   1:  PR[91,2] = PR[90,2] + -10.552;
   1:L PR[91] R[100]mm/sec CNT100;
   1:  PR[91,1] = PR[90,1] + -1.730;
   1:  PR[91,2] = PR[90,2] + -9.704;
   1:L PR[91] R[100]mm/sec CNT100;
   1:  PR[91,1] = PR[90,1] + -0.458;
   1:  PR[91,2] = PR[90,2] + -9.382;
   1:L PR[91] R[100]mm/sec CNT100;
   1:  PR[91,1] = PR[90,1] + 0.617;
   1:L PR[91] R[100]mm/sec CNT100;
   1:  PR[91,1] = PR[90,1] + 1.895;
   1:  PR[91,2] = PR[90,2] + -9.703;
   1:L PR[91] R[100]mm/sec CNT100;
   1:  PR[91,1] = PR[90,1] + 2.818;
   1:  PR[91,2] = PR[90,2] + -10.551;
   1:L PR[91] R[100]mm/sec CNT100;
   1:  PR[91,1] = PR[90,1] + 4.830;
   1:  PR[91,2] = PR[90,2] + -13.079;
   1:L PR[91] R[100]mm/sec CNT100;
   1:  PR[91,1] = PR[90,1] + 7.355;
   1:  PR[91,2] = PR[90,2] + -15.363;
   1:L PR[91] R[100]mm/sec CNT100;
   1:  PR[91,1] = PR[90,1] + 9.557;
   1:  PR[91,2] = PR[90,2] + -16.817;
   1:L PR[91] R[100]mm/sec CNT100;
   1:  PR[91,1] = PR[90,1] + 10.825;
   1:  PR[91,2] = PR[90,2] + -17.449;
   1:L PR[91] R[100]mm/sec CNT100;
   1:  PR[91,1] = PR[90,1] + 12.898;
   1:  PR[91,2] = PR[90,2] + -18.381;
   1:L PR[91] R[100]mm/sec CNT100;
   1:  PR[91,1] = PR[90,1] + 15.573;
   1:  PR[91,2] = PR[90,2] + -19.015;
   1:L PR[91] R[100]mm/sec CNT100;
   1:  PR[91,1] = PR[90,1] + 17.209;
   1:  PR[91,2] = PR[90,2] + -19.446;
   1:L PR[91] R[100]mm/sec CNT100;
   1:  PR[91,1] = PR[90,1] + 18.228;
   1:  PR[91,2] = PR[90,2] + -19.564;
   1:L PR[91] R[100]mm/sec CNT100;
   1:  PR[91,1] = PR[90,1] + 22.320;
   1:  PR[91,2] = PR[90,2] + -19.544;
   1:L PR[91] R[100]mm/sec CNT100;
   1:  PR[91,1] = PR[90,1] + 22.708;
   1:  PR[91,2] = PR[90,2] + -19.528;
   1:L PR[91] R[100]mm/sec CNT100;
   1:  PR[91,1] = PR[90,1] + 27.496;
   1:  PR[91,2] = PR[90,2] + -18.402;
   1:L PR[91] R[100]mm/sec CNT100;
   1:  PR[91,1] = PR[90,1] + 31.736;
   1:  PR[91,2] = PR[90,2] + -16.280;
   1:L PR[91] R[100]mm/sec CNT100;
   1:  PR[91,1] = PR[90,1] + 32.455;
   1:  PR[91,2] = PR[90,2] + -15.698;
   1:L PR[91] R[100]mm/sec CNT100;
   1:  PR[91,1] = PR[90,1] + 35.347;
   1:  PR[91,2] = PR[90,2] + -13.226;
   1:L PR[91] R[100]mm/sec CNT100;
   1:  PR[91,1] = PR[90,1] + 36.249;
   1:  PR[91,2] = PR[90,2] + -12.006;
   1:L PR[91] R[100]mm/sec CNT100;
   1:  PR[91,1] = PR[90,1] + 38.120;
   1:  PR[91,2] = PR[90,2] + -9.367;
   1:L PR[91] R[100]mm/sec CNT100;
   1:  PR[91,1] = PR[90,1] + 38.834;
   1:  PR[91,2] = PR[90,2] + -7.622;
   1:L PR[91] R[100]mm/sec CNT100;
   1:  PR[91,1] = PR[90,1] + 39.865;
   1:  PR[91,2] = PR[90,2] + -5.033;
   1:L PR[91] R[100]mm/sec CNT100;
   1:  PR[91,1] = PR[90,1] + 40.172;
   1:  PR[91,2] = PR[90,2] + -2.721;
   1:L PR[91] R[100]mm/sec CNT100;
   1:  PR[91,1] = PR[90,1] + 40.468;
   1:  PR[91,2] = PR[90,2] + -0.320;
   1:L PR[91] R[100]mm/sec CNT100;
   1:  PR[91,1] = PR[90,1] + 40.178;
   1:  PR[91,2] = PR[90,2] + 1.844;
   1:L PR[91] R[100]mm/sec CNT100;
   1:  PR[91,1] = PR[90,1] + 39.862;
   1:  PR[91,2] = PR[90,2] + 4.417;
   1:L PR[91] R[100]mm/sec CNT100;
   1:  PR[91,1] = PR[90,1] + 38.833;
   1:  PR[91,2] = PR[90,2] + 7.000;
   1:L PR[91] R[100]mm/sec CNT100;
   1:  PR[91,1] = PR[90,1] + 38.120;
   1:  PR[91,2] = PR[90,2] + 8.744;
   1:L PR[91] R[100]mm/sec CNT100;
   1:  PR[91,1] = PR[90,1] + 36.247;
   1:  PR[91,2] = PR[90,2] + 11.384;
   1:L PR[91] R[100]mm/sec CNT100;
   1:  PR[91,1] = PR[90,1] + 35.345;
   1:  PR[91,2] = PR[90,2] + 12.604;
   1:L PR[91] R[100]mm/sec CNT100;
   1:  PR[91,1] = PR[90,1] + 32.451;
   1:  PR[91,2] = PR[90,2] + 15.077;
   1:L PR[91] R[100]mm/sec CNT100;
   1:  PR[91,1] = PR[90,1] + 31.733;
   1:  PR[91,2] = PR[90,2] + 15.658;
   1:L PR[91] R[100]mm/sec CNT100;
   1:  PR[91,1] = PR[90,1] + 27.488;
   1:  PR[91,2] = PR[90,2] + 17.781;
   1:L PR[91] R[100]mm/sec CNT100;
   1:  PR[91,1] = PR[90,1] + 22.979;
   1:  PR[91,2] = PR[90,2] + 18.854;
   1:L PR[91] R[100]mm/sec CNT100;
   1:  PR[91,1] = PR[90,1] + 22.725;
   1:  PR[91,2] = PR[90,2] + 18.904;
   1:L PR[91] R[100]mm/sec CNT100;
   1:  PR[91,1] = PR[90,1] + 22.312;
   1:  PR[91,2] = PR[90,2] + 18.921;
   1:L PR[91] R[100]mm/sec CNT100;
   1:  PR[91,1] = PR[90,1] + 18.222;
   1:  PR[91,2] = PR[90,2] + 18.939;
   1:L PR[91] R[100]mm/sec CNT100;
   1:  PR[91,1] = PR[90,1] + 17.181;
   1:  PR[91,2] = PR[90,2] + 18.819;
   1:L PR[91] R[100]mm/sec CNT100;
   1:  PR[91,1] = PR[90,1] + 14.439;
   1:  PR[91,2] = PR[90,2] + 18.179;
   1:L PR[91] R[100]mm/sec CNT100;
   1:  PR[91,1] = PR[90,1] + 12.914;
   1:  PR[91,2] = PR[90,2] + 17.765;
   1:L PR[91] R[100]mm/sec CNT100;
   1:  PR[91,1] = PR[90,1] + 10.821;
   1:  PR[91,2] = PR[90,2] + 16.824;
   1:L PR[91] R[100]mm/sec CNT100;
   1:  PR[91,1] = PR[90,1] + 9.555;
   1:  PR[91,2] = PR[90,2] + 16.191;
   1:L PR[91] R[100]mm/sec CNT100;
   1:  PR[91,1] = PR[90,1] + 7.337;
   1:  PR[91,2] = PR[90,2] + 14.727;
   1:L PR[91] R[100]mm/sec CNT100;
   1:  PR[91,1] = PR[90,1] + 6.997;
   1:  PR[91,2] = PR[90,2] + 14.436;
   1:L PR[91] R[100]mm/sec CNT100;
   1:  PR[91,1] = PR[90,1] + 4.838;
   1:  PR[91,2] = PR[90,2] + 12.463;
   1:L PR[91] R[100]mm/sec CNT100;
   1:  PR[91,1] = PR[90,1] + 2.867;
   1:  PR[91,2] = PR[90,2] + 9.964;
   1:L PR[91] R[100]mm/sec CNT100;
   1:  PR[91,1] = PR[90,1] + 1.892;
   1:  PR[91,2] = PR[90,2] + 9.079;
   1:L PR[91] R[100]mm/sec CNT100;
   1:  PR[91,1] = PR[90,1] + 0.623;
   1:  PR[91,2] = PR[90,2] + 8.758;
   1:L PR[91] R[100]mm/sec CNT100;
   1:  PR[91,1] = PR[90,1] + -0.452;
   1:L PR[91] R[100]mm/sec CNT100;
   1:  PR[91] = PR[90];
   1:  PR[91,1] = PR[90,1] + -1.625;
   1:  PR[91,2] = PR[90,2] + 9.360;
   1:  PR[91,3] = PR[90,3] + 22.875;
   1:L PR[91] R[100]mm/sec CNT100;
   1:  PR[91,1] = PR[90,1] + -2.543;
   1:  PR[91,2] = PR[90,2] + 10.196;
   1:L PR[91] R[100]mm/sec CNT100;
   1:  PR[91,1] = PR[90,1] + -4.007;
   1:  PR[91,2] = PR[90,2] + 12.033;
   1:L PR[91] R[100]mm/sec CNT100;
   1:  PR[91,1] = PR[90,1] + -4.437;
   1:  PR[91,2] = PR[90,2] + 12.534;
   1:L PR[91] R[100]mm/sec CNT100;
   1:  PR[91,1] = PR[90,1] + -6.783;
   1:  PR[91,2] = PR[90,2] + 14.646;
   1:L PR[91] R[100]mm/sec CNT100;
   1:  PR[91,1] = PR[90,1] + -9.375;
   1:  PR[91,2] = PR[90,2] + 16.350;
   1:L PR[91] R[100]mm/sec CNT100;
   1:  PR[91,1] = PR[90,1] + -9.956;
   1:  PR[91,2] = PR[90,2] + 16.641;
   1:L PR[91] R[100]mm/sec CNT100;
   1:  PR[91,1] = PR[90,1] + -12.537;
   1:  PR[91,2] = PR[90,2] + 17.804;
   1:L PR[91] R[100]mm/sec CNT100;
   1:  PR[91,1] = PR[90,1] + -14.370;
   1:  PR[91,2] = PR[90,2] + 18.238;
   1:L PR[91] R[100]mm/sec CNT100;
   1:  PR[91,1] = PR[90,1] + -16.616;
   1:  PR[91,2] = PR[90,2] + 18.828;
   1:L PR[91] R[100]mm/sec CNT100;
   1:  PR[91,1] = PR[90,1] + -18.071;
   1:  PR[91,2] = PR[90,2] + 18.995;
   1:L PR[91] R[100]mm/sec CNT100;
   1:  PR[91,1] = PR[90,1] + -21.480;
   1:  PR[91,2] = PR[90,2] + 18.979;
   1:L PR[91] R[100]mm/sec CNT100;
   1:  PR[91,1] = PR[90,1] + -22.359;
   1:  PR[91,2] = PR[90,2] + 18.941;
   1:L PR[91] R[100]mm/sec CNT100;
   1:  PR[91,1] = PR[90,1] + -27.198;
   1:  PR[91,2] = PR[90,2] + 17.808;
   1:L PR[91] R[100]mm/sec CNT100;
   1:  PR[91,1] = PR[90,1] + -27.224;
   1:  PR[91,2] = PR[90,2] + 17.799;
   1:L PR[91] R[100]mm/sec CNT100;
   1:  PR[91,1] = PR[90,1] + -31.508;
   1:  PR[91,2] = PR[90,2] + 15.637;
   1:L PR[91] R[100]mm/sec CNT100;
   1:  PR[91,1] = PR[90,1] + -31.793;
   1:  PR[91,2] = PR[90,2] + 15.406;
   1:L PR[91] R[100]mm/sec CNT100;
   1:  PR[91,1] = PR[90,1] + -35.102;
   1:  PR[91,2] = PR[90,2] + 12.583;
   1:L PR[91] R[100]mm/sec CNT100;
   1:  PR[91,1] = PR[90,1] + -35.690;
   1:  PR[91,2] = PR[90,2] + 11.788;
   1:L PR[91] R[100]mm/sec CNT100;
   1:  PR[91,1] = PR[90,1] + -37.860;
   1:  PR[91,2] = PR[90,2] + 8.730;
   1:L PR[91] R[100]mm/sec CNT100;
   1:  PR[91,1] = PR[90,1] + -38.386;
   1:  PR[91,2] = PR[90,2] + 7.439;
   1:L PR[91] R[100]mm/sec CNT100;
   1:  PR[91,1] = PR[90,1] + -39.595;
   1:  PR[91,2] = PR[90,2] + 4.386;
   1:L PR[91] R[100]mm/sec CNT100;
   1:  PR[91,1] = PR[90,1] + -39.833;
   1:  PR[91,2] = PR[90,2] + 2.603;
   1:L PR[91] R[100]mm/sec CNT100;
   1:  PR[91,1] = PR[90,1] + -40.192;
   1:  PR[91,2] = PR[90,2] + -0.304;
   1:L PR[91] R[100]mm/sec CNT100;
   1:  PR[91,1] = PR[90,1] + -39.962;
   1:  PR[91,2] = PR[90,2] + -2.011;
   1:L PR[91] R[100]mm/sec CNT100;
   1:  PR[91,1] = PR[90,1] + -39.593;
   1:  PR[91,2] = PR[90,2] + -5.017;
   1:L PR[91] R[100]mm/sec CNT100;
   1:  PR[91,1] = PR[90,1] + -38.386;
   1:  PR[91,2] = PR[90,2] + -8.063;
   1:L PR[91] R[100]mm/sec CNT100;
   1:  PR[91,1] = PR[90,1] + -37.860;
   1:  PR[91,2] = PR[90,2] + -9.354;
   1:L PR[91] R[100]mm/sec CNT100;
   1:  PR[91,1] = PR[90,1] + -35.690;
   1:  PR[91,2] = PR[90,2] + -12.413;
   1:L PR[91] R[100]mm/sec CNT100;
   1:  PR[91,1] = PR[90,1] + -35.101;
   1:  PR[91,2] = PR[90,2] + -13.207;
   1:L PR[91] R[100]mm/sec CNT100;
   1:  PR[91,1] = PR[90,1] + -31.793;
   1:  PR[91,2] = PR[90,2] + -16.030;
   1:L PR[91] R[100]mm/sec CNT100;
   1:  PR[91,1] = PR[90,1] + -31.508;
   1:  PR[91,2] = PR[90,2] + -16.261;
   1:L PR[91] R[100]mm/sec CNT100;
   1:  PR[91,1] = PR[90,1] + -27.224;
   1:  PR[91,2] = PR[90,2] + -18.423;
   1:L PR[91] R[100]mm/sec CNT100;
   1:  PR[91,1] = PR[90,1] + -27.194;
   1:  PR[91,2] = PR[90,2] + -18.434;
   1:L PR[91] R[100]mm/sec CNT100;
   1:  PR[91,1] = PR[90,1] + -22.977;
   1:  PR[91,2] = PR[90,2] + -19.446;
   1:L PR[91] R[100]mm/sec CNT100;
   1:  PR[91,1] = PR[90,1] + -22.382;
   1:  PR[91,2] = PR[90,2] + -19.564;
   1:L PR[91] R[100]mm/sec CNT100;
   1:  PR[91,1] = PR[90,1] + -21.480;
   1:  PR[91,2] = PR[90,2] + -19.603;
   1:L PR[91] R[100]mm/sec CNT100;
   1:  PR[91,1] = PR[90,1] + -18.071;
   1:  PR[91,2] = PR[90,2] + -19.619;
   1:L PR[91] R[100]mm/sec CNT100;
   1:  PR[91,1] = PR[90,1] + -16.595;
   1:  PR[91,2] = PR[90,2] + -19.450;
   1:L PR[91] R[100]mm/sec CNT100;
   1:  PR[91,1] = PR[90,1] + -14.455;
   1:  PR[91,2] = PR[90,2] + -18.953;
   1:L PR[91] R[100]mm/sec CNT100;
   1:  PR[91,1] = PR[90,1] + -12.559;
   1:  PR[91,2] = PR[90,2] + -18.438;
   1:L PR[91] R[100]mm/sec CNT100;
   1:  PR[91,1] = PR[90,1] + -9.956;
   1:  PR[91,2] = PR[90,2] + -17.265;
   1:L PR[91] R[100]mm/sec CNT100;
   1:  PR[91,1] = PR[90,1] + -9.375;
   1:  PR[91,2] = PR[90,2] + -16.974;
   1:L PR[91] R[100]mm/sec CNT100;
   1:  PR[91,1] = PR[90,1] + -6.778;
   1:  PR[91,2] = PR[90,2] + -15.266;
   1:L PR[91] R[100]mm/sec CNT100;
   1:  PR[91,1] = PR[90,1] + -4.421;
   1:  PR[91,2] = PR[90,2] + -13.143;
   1:L PR[91] R[100]mm/sec CNT100;
   1:  PR[91,1] = PR[90,1] + -4.010;
   1:  PR[91,2] = PR[90,2] + -12.660;
   1:L PR[91] R[100]mm/sec CNT100;
   1:  PR[91,1] = PR[90,1] + -2.559;
   1:  PR[91,2] = PR[90,2] + -10.827;
   1:L PR[91] R[100]mm/sec CNT100;
   1:  PR[91,1] = PR[90,1] + -2.107;
   1:  PR[91,2] = PR[90,2] + -10.408;
   1:L PR[91] R[100]mm/sec CNT100;
   1:  PR[91,1] = PR[90,1] + -1.599;
   1:  PR[91,2] = PR[90,2] + -9.979;
   1:L PR[91] R[100]mm/sec CNT100;
   1:  PR[91,1] = PR[90,1] + -0.366;
   1:  PR[91,2] = PR[90,2] + -9.671;
   1:L PR[91] R[100]mm/sec CNT100;
   1:  PR[91,1] = PR[90,1] + 0.518;
   1:L PR[91] R[100]mm/sec CNT100;
   1:  PR[91,1] = PR[90,1] + 1.789;
   1:  PR[91,2] = PR[90,2] + -9.983;
   1:L PR[91] R[100]mm/sec CNT100;
   1:  PR[91,1] = PR[90,1] + 2.707;
   1:  PR[91,2] = PR[90,2] + -10.818;
   1:L PR[91] R[100]mm/sec CNT100;
   1:  PR[91,1] = PR[90,1] + 4.190;
   1:  PR[91,2] = PR[90,2] + -12.679;
   1:L PR[91] R[100]mm/sec CNT100;
   1:  PR[91,1] = PR[90,1] + 4.604;
   1:  PR[91,2] = PR[90,2] + -13.165;
   1:L PR[91] R[100]mm/sec CNT100;
   1:  PR[91,1] = PR[90,1] + 6.958;
   1:  PR[91,2] = PR[90,2] + -15.287;
   1:L PR[91] R[100]mm/sec CNT100;
   1:  PR[91,1] = PR[90,1] + 9.528;
   1:  PR[91,2] = PR[90,2] + -16.975;
   1:L PR[91] R[100]mm/sec CNT100;
   1:  PR[91,1] = PR[90,1] + 10.108;
   1:  PR[91,2] = PR[90,2] + -17.265;
   1:L PR[91] R[100]mm/sec CNT100;
   1:  PR[91,1] = PR[90,1] + 12.688;
   1:  PR[91,2] = PR[90,2] + -18.424;
   1:L PR[91] R[100]mm/sec CNT100;
   1:  PR[91,1] = PR[90,1] + 14.520;
   1:  PR[91,2] = PR[90,2] + -18.859;
   1:L PR[91] R[100]mm/sec CNT100;
   1:  PR[91,1] = PR[90,1] + 16.772;
   1:  PR[91,2] = PR[90,2] + -19.452;
   1:L PR[91] R[100]mm/sec CNT100;
   1:  PR[91,1] = PR[90,1] + 18.224;
   1:  PR[91,2] = PR[90,2] + -19.619;
   1:L PR[91] R[100]mm/sec CNT100;
   1:  PR[91,1] = PR[90,1] + 21.633;
   1:  PR[91,2] = PR[90,2] + -19.603;
   1:L PR[91] R[100]mm/sec CNT100;
   1:  PR[91,1] = PR[90,1] + 22.509;
   1:  PR[91,2] = PR[90,2] + -19.566;
   1:L PR[91] R[100]mm/sec CNT100;
   1:  PR[91,1] = PR[90,1] + 27.353;
   1:  PR[91,2] = PR[90,2] + -18.431;
   1:L PR[91] R[100]mm/sec CNT100;
   1:  PR[91,1] = PR[90,1] + 27.381;
   1:  PR[91,2] = PR[90,2] + -18.421;
   1:L PR[91] R[100]mm/sec CNT100;
   1:  PR[91,1] = PR[90,1] + 31.664;
   1:  PR[91,2] = PR[90,2] + -16.264;
   1:L PR[91] R[100]mm/sec CNT100;
   1:  PR[91,1] = PR[90,1] + 31.949;
   1:  PR[91,2] = PR[90,2] + -16.034;
   1:L PR[91] R[100]mm/sec CNT100;
   1:  PR[91,1] = PR[90,1] + 35.258;
   1:  PR[91,2] = PR[90,2] + -13.206;
   1:L PR[91] R[100]mm/sec CNT100;
   1:  PR[91,1] = PR[90,1] + 35.846;
   1:  PR[91,2] = PR[90,2] + -12.410;
   1:L PR[91] R[100]mm/sec CNT100;
   1:  PR[91,1] = PR[90,1] + 38.014;
   1:  PR[91,2] = PR[90,2] + -9.352;
   1:L PR[91] R[100]mm/sec CNT100;
   1:  PR[91,1] = PR[90,1] + 39.752;
   1:  PR[91,2] = PR[90,2] + -5.024;
   1:L PR[91] R[100]mm/sec CNT100;
   1:  PR[91,1] = PR[90,1] + 39.990;
   1:  PR[91,2] = PR[90,2] + -3.239;
   1:L PR[91] R[100]mm/sec CNT100;
   1:  PR[91,1] = PR[90,1] + 40.349;
   1:  PR[91,2] = PR[90,2] + -0.320;
   1:L PR[91] R[100]mm/sec CNT100;
   1:  PR[91,1] = PR[90,1] + 40.119;
   1:  PR[91,2] = PR[90,2] + 1.392;
   1:L PR[91] R[100]mm/sec CNT100;
   1:  PR[91,1] = PR[90,1] + 39.749;
   1:  PR[91,2] = PR[90,2] + 4.407;
   1:L PR[91] R[100]mm/sec CNT100;
   1:  PR[91,1] = PR[90,1] + 38.013;
   1:  PR[91,2] = PR[90,2] + 8.730;
   1:L PR[91] R[100]mm/sec CNT100;
   1:  PR[91,1] = PR[90,1] + 35.844;
   1:  PR[91,2] = PR[90,2] + 11.789;
   1:L PR[91] R[100]mm/sec CNT100;
   1:  PR[91,1] = PR[90,1] + 35.256;
   1:  PR[91,2] = PR[90,2] + 12.584;
   1:L PR[91] R[100]mm/sec CNT100;
   1:  PR[91,1] = PR[90,1] + 31.944;
   1:  PR[91,2] = PR[90,2] + 15.413;
   1:L PR[91] R[100]mm/sec CNT100;
   1:  PR[91,1] = PR[90,1] + 31.660;
   1:  PR[91,2] = PR[90,2] + 15.643;
   1:L PR[91] R[100]mm/sec CNT100;
   1:  PR[91,1] = PR[90,1] + 27.374;
   1:  PR[91,2] = PR[90,2] + 17.799;
   1:L PR[91] R[100]mm/sec CNT100;
   1:  PR[91,1] = PR[90,1] + 27.343;
   1:  PR[91,2] = PR[90,2] + 17.811;
   1:L PR[91] R[100]mm/sec CNT100;
   1:  PR[91,1] = PR[90,1] + 23.123;
   1:  PR[91,2] = PR[90,2] + 18.824;
   1:L PR[91] R[100]mm/sec CNT100;
   1:  PR[91,1] = PR[90,1] + 22.527;
   1:  PR[91,2] = PR[90,2] + 18.942;
   1:L PR[91] R[100]mm/sec CNT100;
   1:  PR[91,1] = PR[90,1] + 21.627;
   1:  PR[91,2] = PR[90,2] + 18.980;
   1:L PR[91] R[100]mm/sec CNT100;
   1:  PR[91,1] = PR[90,1] + 18.218;
   1:  PR[91,2] = PR[90,2] + 18.994;
   1:L PR[91] R[100]mm/sec CNT100;
   1:  PR[91,1] = PR[90,1] + 16.746;
   1:  PR[91,2] = PR[90,2] + 18.825;
   1:L PR[91] R[100]mm/sec CNT100;
   1:  PR[91,1] = PR[90,1] + 14.607;
   1:  PR[91,2] = PR[90,2] + 18.326;
   1:L PR[91] R[100]mm/sec CNT100;
   1:  PR[91,1] = PR[90,1] + 12.706;
   1:  PR[91,2] = PR[90,2] + 17.808;
   1:L PR[91] R[100]mm/sec CNT100;
   1:  PR[91,1] = PR[90,1] + 10.107;
   1:  PR[91,2] = PR[90,2] + 16.640;
   1:L PR[91] R[100]mm/sec CNT100;
   1:  PR[91,1] = PR[90,1] + 9.527;
   1:  PR[91,2] = PR[90,2] + 16.351;
   1:L PR[91] R[100]mm/sec CNT100;
   1:  PR[91,1] = PR[90,1] + 6.962;
   1:  PR[91,2] = PR[90,2] + 14.667;
   1:L PR[91] R[100]mm/sec CNT100;
   1:  PR[91,1] = PR[90,1] + 4.591;
   1:  PR[91,2] = PR[90,2] + 12.531;
   1:L PR[91] R[100]mm/sec CNT100;
   1:  PR[91,1] = PR[90,1] + 4.554;
   1:  PR[91,2] = PR[90,2] + 12.492;
   1:L PR[91] R[100]mm/sec CNT100;
   1:  PR[91,1] = PR[90,1] + 2.769;
   1:  PR[91,2] = PR[90,2] + 10.224;
   1:L PR[91] R[100]mm/sec CNT100;
   1:  PR[91,1] = PR[90,1] + 2.592;
   1:  PR[91,2] = PR[90,2] + 10.088;
   1:L PR[91] R[100]mm/sec CNT100;
   1:  PR[91,1] = PR[90,1] + 2.279;
   1:  PR[91,2] = PR[90,2] + 9.789;
   1:L PR[91] R[100]mm/sec CNT100;
   1:  PR[91,1] = PR[90,1] + 1.763;
   1:  PR[91,2] = PR[90,2] + 9.354;
   1:L PR[91] R[100]mm/sec CNT100;
   1:  PR[91,1] = PR[90,1] + 0.530;
   1:  PR[91,2] = PR[90,2] + 9.047;
   1:L PR[91] R[100]mm/sec CNT100;
   1:  PR[91,1] = PR[90,1] + -0.352;
   1:L PR[91] R[100]mm/sec CNT100;
   1:  PR[91] = PR[90];
   1:  PR[91,1] = PR[90,1] + -1.514;
   1:  PR[91,2] = PR[90,2] + 9.639;
   1:  PR[91,3] = PR[90,3] + 23.485;
   1:L PR[91] R[100]mm/sec CNT100;
   1:  PR[91,1] = PR[90,1] + -2.434;
   1:  PR[91,2] = PR[90,2] + 10.459;
   1:L PR[91] R[100]mm/sec CNT100;
   1:  PR[91,1] = PR[90,1] + -3.410;
   1:  PR[91,2] = PR[90,2] + 11.680;
   1:L PR[91] R[100]mm/sec CNT100;
   1:  PR[91,1] = PR[90,1] + -4.067;
   1:  PR[91,2] = PR[90,2] + 12.470;
   1:L PR[91] R[100]mm/sec CNT100;
   1:  PR[91,1] = PR[90,1] + -4.215;
   1:  PR[91,2] = PR[90,2] + 12.625;
   1:L PR[91] R[100]mm/sec CNT100;
   1:  PR[91,1] = PR[90,1] + -6.555;
   1:  PR[91,2] = PR[90,2] + 14.723;
   1:L PR[91] R[100]mm/sec CNT100;
   1:  PR[91,1] = PR[90,1] + -9.313;
   1:  PR[91,2] = PR[90,2] + 16.490;
   1:L PR[91] R[100]mm/sec CNT100;
   1:  PR[91,1] = PR[90,1] + -12.328;
   1:  PR[91,2] = PR[90,2] + 17.848;
   1:L PR[91] R[100]mm/sec CNT100;
   1:  PR[91,1] = PR[90,1] + -13.319;
   1:  PR[91,2] = PR[90,2] + 18.083;
   1:L PR[91] R[100]mm/sec CNT100;
   1:  PR[91,1] = PR[90,1] + -16.179;
   1:  PR[91,2] = PR[90,2] + 18.834;
   1:L PR[91] R[100]mm/sec CNT100;
   1:  PR[91,1] = PR[90,1] + -18.067;
   1:  PR[91,2] = PR[90,2] + 19.050;
   1:L PR[91] R[100]mm/sec CNT100;
   1:  PR[91,1] = PR[90,1] + -20.795;
   1:  PR[91,2] = PR[90,2] + 19.037;
   1:L PR[91] R[100]mm/sec CNT100;
   1:  PR[91,1] = PR[90,1] + -22.161;
   1:  PR[91,2] = PR[90,2] + 18.979;
   1:L PR[91] R[100]mm/sec CNT100;
   1:  PR[91,1] = PR[90,1] + -26.109;
   1:  PR[91,2] = PR[90,2] + 18.049;
   1:L PR[91] R[100]mm/sec CNT100;
   1:  PR[91,1] = PR[90,1] + -26.826;
   1:  PR[91,2] = PR[90,2] + 17.900;
   1:L PR[91] R[100]mm/sec CNT100;
   1:  PR[91,1] = PR[90,1] + -27.197;
   1:  PR[91,2] = PR[90,2] + 17.765;
   1:L PR[91] R[100]mm/sec CNT100;
   1:  PR[91,1] = PR[90,1] + -31.416;
   1:  PR[91,2] = PR[90,2] + 15.631;
   1:L PR[91] R[100]mm/sec CNT100;
   1:  PR[91,1] = PR[90,1] + -35.012;
   1:  PR[91,2] = PR[90,2] + 12.563;
   1:L PR[91] R[100]mm/sec CNT100;
   1:  PR[91,1] = PR[90,1] + -35.287;
   1:  PR[91,2] = PR[90,2] + 12.192;
   1:L PR[91] R[100]mm/sec CNT100;
   1:  PR[91,1] = PR[90,1] + -37.753;
   1:  PR[91,2] = PR[90,2] + 8.716;
   1:L PR[91] R[100]mm/sec CNT100;
   1:  PR[91,1] = PR[90,1] + -39.482;
   1:  PR[91,2] = PR[90,2] + 4.377;
   1:L PR[91] R[100]mm/sec CNT100;
   1:  PR[91,1] = PR[90,1] + -39.650;
   1:  PR[91,2] = PR[90,2] + 3.118;
   1:L PR[91] R[100]mm/sec CNT100;
   1:  PR[91,1] = PR[90,1] + -40.073;
   1:  PR[91,2] = PR[90,2] + -0.304;
   1:L PR[91] R[100]mm/sec CNT100;
   1:  PR[91,1] = PR[90,1] + -39.904;
   1:  PR[91,2] = PR[90,2] + -1.560;
   1:L PR[91] R[100]mm/sec CNT100;
   1:  PR[91,1] = PR[90,1] + -39.479;
   1:  PR[91,2] = PR[90,2] + -5.009;
   1:L PR[91] R[100]mm/sec CNT100;
   1:  PR[91,1] = PR[90,1] + -38.095;
   1:  PR[91,2] = PR[90,2] + -8.505;
   1:L PR[91] R[100]mm/sec CNT100;
   1:  PR[91,1] = PR[90,1] + -37.756;
   1:  PR[91,2] = PR[90,2] + -9.336;
   1:L PR[91] R[100]mm/sec CNT100;
   1:  PR[91,1] = PR[90,1] + -35.286;
   1:  PR[91,2] = PR[90,2] + -12.816;
   1:L PR[91] R[100]mm/sec CNT100;
   1:  PR[91,1] = PR[90,1] + -35.012;
   1:  PR[91,2] = PR[90,2] + -13.187;
   1:L PR[91] R[100]mm/sec CNT100;
   1:  PR[91,1] = PR[90,1] + -31.415;
   1:  PR[91,2] = PR[90,2] + -16.255;
   1:L PR[91] R[100]mm/sec CNT100;
   1:  PR[91,1] = PR[90,1] + -27.197;
   1:  PR[91,2] = PR[90,2] + -18.389;
   1:L PR[91] R[100]mm/sec CNT100;
   1:  PR[91,1] = PR[90,1] + -26.805;
   1:  PR[91,2] = PR[90,2] + -18.532;
   1:L PR[91] R[100]mm/sec CNT100;
   1:  PR[91,1] = PR[90,1] + -23.123;
   1:  PR[91,2] = PR[90,2] + -19.415;
   1:L PR[91] R[100]mm/sec CNT100;
   1:  PR[91,1] = PR[90,1] + -22.186;
   1:  PR[91,2] = PR[90,2] + -19.602;
   1:L PR[91] R[100]mm/sec CNT100;
   1:  PR[91,1] = PR[90,1] + -20.795;
   1:  PR[91,2] = PR[90,2] + -19.661;
   1:L PR[91] R[100]mm/sec CNT100;
   1:  PR[91,1] = PR[90,1] + -18.067;
   1:  PR[91,2] = PR[90,2] + -19.674;
   1:L PR[91] R[100]mm/sec CNT100;
   1:  PR[91,1] = PR[90,1] + -16.159;
   1:  PR[91,2] = PR[90,2] + -19.455;
   1:L PR[91] R[100]mm/sec CNT100;
   1:  PR[91,1] = PR[90,1] + -14.622;
   1:  PR[91,2] = PR[90,2] + -19.099;
   1:L PR[91] R[100]mm/sec CNT100;
   1:  PR[91,1] = PR[90,1] + -12.350;
   1:  PR[91,2] = PR[90,2] + -18.482;
   1:L PR[91] R[100]mm/sec CNT100;
   1:  PR[91,1] = PR[90,1] + -9.313;
   1:  PR[91,2] = PR[90,2] + -17.113;
   1:L PR[91] R[100]mm/sec CNT100;
   1:  PR[91,1] = PR[90,1] + -6.576;
   1:  PR[91,2] = PR[90,2] + -15.363;
   1:L PR[91] R[100]mm/sec CNT100;
   1:  PR[91,1] = PR[90,1] + -6.379;
   1:  PR[91,2] = PR[90,2] + -15.198;
   1:L PR[91] R[100]mm/sec CNT100;
   1:  PR[91,1] = PR[90,1] + -4.216;
   1:  PR[91,2] = PR[90,2] + -13.248;
   1:L PR[91] R[100]mm/sec CNT100;
   1:  PR[91,1] = PR[90,1] + -3.407;
   1:  PR[91,2] = PR[90,2] + -12.300;
   1:L PR[91] R[100]mm/sec CNT100;
   1:  PR[91,1] = PR[90,1] + -2.456;
   1:  PR[91,2] = PR[90,2] + -11.098;
   1:L PR[91] R[100]mm/sec CNT100;
   1:  PR[91,1] = PR[90,1] + -2.127;
   1:  PR[91,2] = PR[90,2] + -10.792;
   1:L PR[91] R[100]mm/sec CNT100;
   1:  PR[91,1] = PR[90,1] + -1.497;
   1:  PR[91,2] = PR[90,2] + -10.260;
   1:L PR[91] R[100]mm/sec CNT100;
   1:  PR[91,1] = PR[90,1] + -0.273;
   1:  PR[91,2] = PR[90,2] + -9.959;
   1:L PR[91] R[100]mm/sec CNT100;
   1:  PR[91,1] = PR[90,1] + 0.424;
   1:L PR[91] R[100]mm/sec CNT100;
   1:  PR[91,1] = PR[90,1] + 1.678;
   1:  PR[91,2] = PR[90,2] + -10.263;
   1:L PR[91] R[100]mm/sec CNT100;
   1:  PR[91,1] = PR[90,1] + 2.600;
   1:  PR[91,2] = PR[90,2] + -11.082;
   1:L PR[91] R[100]mm/sec CNT100;
   1:  PR[91,1] = PR[90,1] + 3.581;
   1:  PR[91,2] = PR[90,2] + -12.311;
   1:L PR[91] R[100]mm/sec CNT100;
   1:  PR[91,1] = PR[90,1] + 4.395;
   1:  PR[91,2] = PR[90,2] + -13.268;
   1:L PR[91] R[100]mm/sec CNT100;
   1:  PR[91,1] = PR[90,1] + 6.705;
   1:  PR[91,2] = PR[90,2] + -15.346;
   1:L PR[91] R[100]mm/sec CNT100;
   1:  PR[91,1] = PR[90,1] + 9.466;
   1:  PR[91,2] = PR[90,2] + -17.114;
   1:L PR[91] R[100]mm/sec CNT100;
   1:  PR[91,1] = PR[90,1] + 12.477;
   1:  PR[91,2] = PR[90,2] + -18.467;
   1:L PR[91] R[100]mm/sec CNT100;
   1:  PR[91,1] = PR[90,1] + 13.467;
   1:  PR[91,2] = PR[90,2] + -18.702;
   1:L PR[91] R[100]mm/sec CNT100;
   1:  PR[91,1] = PR[90,1] + 16.335;
   1:  PR[91,2] = PR[90,2] + -19.457;
   1:L PR[91] R[100]mm/sec CNT100;
   1:  PR[91,1] = PR[90,1] + 18.219;
   1:  PR[91,2] = PR[90,2] + -19.674;
   1:L PR[91] R[100]mm/sec CNT100;
   1:  PR[91,1] = PR[90,1] + 20.947;
   1:  PR[91,2] = PR[90,2] + -19.661;
   1:L PR[91] R[100]mm/sec CNT100;
   1:  PR[91,1] = PR[90,1] + 22.309;
   1:  PR[91,2] = PR[90,2] + -19.604;
   1:L PR[91] R[100]mm/sec CNT100;
   1:  PR[91,1] = PR[90,1] + 26.258;
   1:  PR[91,2] = PR[90,2] + -18.673;
   1:L PR[91] R[100]mm/sec CNT100;
   1:  PR[91,1] = PR[90,1] + 26.979;
   1:  PR[91,2] = PR[90,2] + -18.523;
   1:L PR[91] R[100]mm/sec CNT100;
   1:  PR[91,1] = PR[90,1] + 27.352;
   1:  PR[91,2] = PR[90,2] + -18.388;
   1:L PR[91] R[100]mm/sec CNT100;
   1:  PR[91,1] = PR[90,1] + 31.572;
   1:  PR[91,2] = PR[90,2] + -16.258;
   1:L PR[91] R[100]mm/sec CNT100;
   1:  PR[91,1] = PR[90,1] + 35.168;
   1:  PR[91,2] = PR[90,2] + -13.185;
   1:L PR[91] R[100]mm/sec CNT100;
   1:  PR[91,1] = PR[90,1] + 35.443;
   1:  PR[91,2] = PR[90,2] + -12.814;
   1:L PR[91] R[100]mm/sec CNT100;
   1:  PR[91,1] = PR[90,1] + 37.910;
   1:  PR[91,2] = PR[90,2] + -9.335;
   1:L PR[91] R[100]mm/sec CNT100;
   1:  PR[91,1] = PR[90,1] + 39.639;
   1:  PR[91,2] = PR[90,2] + -5.017;
   1:L PR[91] R[100]mm/sec CNT100;
   1:  PR[91,1] = PR[90,1] + 39.807;
   1:  PR[91,2] = PR[90,2] + -3.756;
   1:L PR[91] R[100]mm/sec CNT100;
   1:  PR[91,1] = PR[90,1] + 40.229;
   1:  PR[91,2] = PR[90,2] + -0.320;
   1:L PR[91] R[100]mm/sec CNT100;
   1:  PR[91,1] = PR[90,1] + 40.061;
   1:  PR[91,2] = PR[90,2] + 0.940;
   1:L PR[91] R[100]mm/sec CNT100;
   1:  PR[91,1] = PR[90,1] + 39.636;
   1:  PR[91,2] = PR[90,2] + 4.401;
   1:L PR[91] R[100]mm/sec CNT100;
   1:  PR[91,1] = PR[90,1] + 37.909;
   1:  PR[91,2] = PR[90,2] + 8.712;
   1:L PR[91] R[100]mm/sec CNT100;
   1:  PR[91,1] = PR[90,1] + 35.440;
   1:  PR[91,2] = PR[90,2] + 12.193;
   1:L PR[91] R[100]mm/sec CNT100;
   1:  PR[91,1] = PR[90,1] + 35.166;
   1:  PR[91,2] = PR[90,2] + 12.564;
   1:L PR[91] R[100]mm/sec CNT100;
   1:  PR[91,1] = PR[90,1] + 31.567;
   1:  PR[91,2] = PR[90,2] + 15.637;
   1:L PR[91] R[100]mm/sec CNT100;
   1:  PR[91,1] = PR[90,1] + 27.346;
   1:  PR[91,2] = PR[90,2] + 17.766;
   1:L PR[91] R[100]mm/sec CNT100;
   1:  PR[91,1] = PR[90,1] + 26.951;
   1:  PR[91,2] = PR[90,2] + 17.909;
   1:L PR[91] R[100]mm/sec CNT100;
   1:  PR[91,1] = PR[90,1] + 23.267;
   1:  PR[91,2] = PR[90,2] + 18.794;
   1:L PR[91] R[100]mm/sec CNT100;
   1:  PR[91,1] = PR[90,1] + 22.329;
   1:  PR[91,2] = PR[90,2] + 18.980;
   1:L PR[91] R[100]mm/sec CNT100;
   1:  PR[91,1] = PR[90,1] + 20.941;
   1:  PR[91,2] = PR[90,2] + 19.038;
   1:L PR[91] R[100]mm/sec CNT100;
   1:  PR[91,1] = PR[90,1] + 18.214;
   1:  PR[91,2] = PR[90,2] + 19.050;
   1:L PR[91] R[100]mm/sec CNT100;
   1:  PR[91,1] = PR[90,1] + 16.310;
   1:  PR[91,2] = PR[90,2] + 18.830;
   1:L PR[91] R[100]mm/sec CNT100;
   1:  PR[91,1] = PR[90,1] + 14.775;
   1:  PR[91,2] = PR[90,2] + 18.472;
   1:L PR[91] R[100]mm/sec CNT100;
   1:  PR[91,1] = PR[90,1] + 12.497;
   1:  PR[91,2] = PR[90,2] + 17.852;
   1:L PR[91] R[100]mm/sec CNT100;
   1:  PR[91,1] = PR[90,1] + 9.466;
   1:  PR[91,2] = PR[90,2] + 16.490;
   1:L PR[91] R[100]mm/sec CNT100;
   1:  PR[91,1] = PR[90,1] + 6.734;
   1:  PR[91,2] = PR[90,2] + 14.743;
   1:L PR[91] R[100]mm/sec CNT100;
   1:  PR[91,1] = PR[90,1] + 4.396;
   1:  PR[91,2] = PR[90,2] + 12.646;
   1:L PR[91] R[100]mm/sec CNT100;
   1:  PR[91,1] = PR[90,1] + 4.260;
   1:  PR[91,2] = PR[90,2] + 12.504;
   1:L PR[91] R[100]mm/sec CNT100;
   1:  PR[91,1] = PR[90,1] + 2.742;
   1:  PR[91,2] = PR[90,2] + 10.574;
   1:L PR[91] R[100]mm/sec CNT100;
   1:  PR[91,1] = PR[90,1] + 2.284;
   1:  PR[91,2] = PR[90,2] + 10.161;
   1:L PR[91] R[100]mm/sec CNT100;
   1:  PR[91,1] = PR[90,1] + 1.661;
   1:  PR[91,2] = PR[90,2] + 9.636;
   1:L PR[91] R[100]mm/sec CNT100;
   1:  PR[91,1] = PR[90,1] + 0.437;
   1:  PR[91,2] = PR[90,2] + 9.335;
   1:L PR[91] R[100]mm/sec CNT100;
   1:  PR[91,1] = PR[90,1] + -0.258;
   1:L PR[91] R[100]mm/sec CNT100;
   1:  PR[91] = PR[90];
   1:  PR[91,1] = PR[90,1] + -1.401;
   1:  PR[91,2] = PR[90,2] + 9.919;
   1:  PR[91,3] = PR[90,3] + 24.095;
   1:L PR[91] R[100]mm/sec CNT100;
   1:  PR[91,1] = PR[90,1] + -2.322;
   1:  PR[91,2] = PR[90,2] + 10.715;
   1:L PR[91] R[100]mm/sec CNT100;
   1:  PR[91,1] = PR[90,1] + -3.778;
   1:  PR[91,2] = PR[90,2] + 12.487;
   1:L PR[91] R[100]mm/sec CNT100;
   1:  PR[91,1] = PR[90,1] + -4.025;
   1:  PR[91,2] = PR[90,2] + 12.745;
   1:L PR[91] R[100]mm/sec CNT100;
   1:  PR[91,1] = PR[90,1] + -6.030;
   1:  PR[91,2] = PR[90,2] + 14.552;
   1:L PR[91] R[100]mm/sec CNT100;
   1:  PR[91,1] = PR[90,1] + -6.319;
   1:  PR[91,2] = PR[90,2] + 14.797;
   1:L PR[91] R[100]mm/sec CNT100;
   1:  PR[91,1] = PR[90,1] + -9.021;
   1:  PR[91,2] = PR[90,2] + 16.529;
   1:L PR[91] R[100]mm/sec CNT100;
   1:  PR[91,1] = PR[90,1] + -12.128;
   1:  PR[91,2] = PR[90,2] + 17.897;
   1:L PR[91] R[100]mm/sec CNT100;
   1:  PR[91,1] = PR[90,1] + -15.741;
   1:  PR[91,2] = PR[90,2] + 18.839;
   1:L PR[91] R[100]mm/sec CNT100;
   1:  PR[91,1] = PR[90,1] + -18.064;
   1:  PR[91,2] = PR[90,2] + 19.105;
   1:L PR[91] R[100]mm/sec CNT100;
   1:  PR[91,1] = PR[90,1] + -20.110;
   1:  PR[91,2] = PR[90,2] + 19.096;
   1:L PR[91] R[100]mm/sec CNT100;
   1:  PR[91,1] = PR[90,1] + -21.964;
   1:  PR[91,2] = PR[90,2] + 19.017;
   1:L PR[91] R[100]mm/sec CNT100;
   1:  PR[91,1] = PR[90,1] + -25.192;
   1:  PR[91,2] = PR[90,2] + 18.256;
   1:L PR[91] R[100]mm/sec CNT100;
   1:  PR[91,1] = PR[90,1] + -26.437;
   1:  PR[91,2] = PR[90,2] + 17.998;
   1:L PR[91] R[100]mm/sec CNT100;
   1:  PR[91,1] = PR[90,1] + -27.172;
   1:  PR[91,2] = PR[90,2] + 17.731;
   1:L PR[91] R[100]mm/sec CNT100;
   1:  PR[91,1] = PR[90,1] + -30.981;
   1:  PR[91,2] = PR[90,2] + 15.804;
   1:L PR[91] R[100]mm/sec CNT100;
   1:  PR[91,1] = PR[90,1] + -31.213;
   1:  PR[91,2] = PR[90,2] + 15.675;
   1:L PR[91] R[100]mm/sec CNT100;
   1:  PR[91,1] = PR[90,1] + -34.914;
   1:  PR[91,2] = PR[90,2] + 12.549;
   1:L PR[91] R[100]mm/sec CNT100;
   1:  PR[91,1] = PR[90,1] + -37.648;
   1:  PR[91,2] = PR[90,2] + 8.699;
   1:L PR[91] R[100]mm/sec CNT100;
   1:  PR[91,1] = PR[90,1] + -39.367;
   1:  PR[91,2] = PR[90,2] + 4.375;
   1:L PR[91] R[100]mm/sec CNT100;
   1:  PR[91,1] = PR[90,1] + -39.954;
   1:  PR[91,2] = PR[90,2] + -0.312;
   1:L PR[91] R[100]mm/sec CNT100;
   1:  PR[91,1] = PR[90,1] + -39.367;
   1:  PR[91,2] = PR[90,2] + -5.000;
   1:L PR[91] R[100]mm/sec CNT100;
   1:  PR[91,1] = PR[90,1] + -37.804;
   1:  PR[91,2] = PR[90,2] + -8.945;
   1:L PR[91] R[100]mm/sec CNT100;
   1:  PR[91,1] = PR[90,1] + -37.652;
   1:  PR[91,2] = PR[90,2] + -9.318;
   1:L PR[91] R[100]mm/sec CNT100;
   1:  PR[91,1] = PR[90,1] + -34.913;
   1:  PR[91,2] = PR[90,2] + -13.175;
   1:L PR[91] R[100]mm/sec CNT100;
   1:  PR[91,1] = PR[90,1] + -31.388;
   1:  PR[91,2] = PR[90,2] + -16.169;
   1:L PR[91] R[100]mm/sec CNT100;
   1:  PR[91,1] = PR[90,1] + -31.237;
   1:  PR[91,2] = PR[90,2] + -16.286;
   1:L PR[91] R[100]mm/sec CNT100;
   1:  PR[91,1] = PR[90,1] + -30.981;
   1:  PR[91,2] = PR[90,2] + -16.428;
   1:L PR[91] R[100]mm/sec CNT100;
   1:  PR[91,1] = PR[90,1] + -27.171;
   1:  PR[91,2] = PR[90,2] + -18.355;
   1:L PR[91] R[100]mm/sec CNT100;
   1:  PR[91,1] = PR[90,1] + -26.416;
   1:  PR[91,2] = PR[90,2] + -18.630;
   1:L PR[91] R[100]mm/sec CNT100;
   1:  PR[91,1] = PR[90,1] + -23.270;
   1:  PR[91,2] = PR[90,2] + -19.385;
   1:L PR[91] R[100]mm/sec CNT100;
   1:  PR[91,1] = PR[90,1] + -21.989;
   1:  PR[91,2] = PR[90,2] + -19.640;
   1:L PR[91] R[100]mm/sec CNT100;
   1:  PR[91,1] = PR[90,1] + -20.110;
   1:  PR[91,2] = PR[90,2] + -19.720;
   1:L PR[91] R[100]mm/sec CNT100;
   1:  PR[91,1] = PR[90,1] + -18.063;
   1:  PR[91,2] = PR[90,2] + -19.729;
   1:L PR[91] R[100]mm/sec CNT100;
   1:  PR[91,1] = PR[90,1] + -15.722;
   1:  PR[91,2] = PR[90,2] + -19.461;
   1:L PR[91] R[100]mm/sec CNT100;
   1:  PR[91,1] = PR[90,1] + -14.790;
   1:  PR[91,2] = PR[90,2] + -19.245;
   1:L PR[91] R[100]mm/sec CNT100;
   1:  PR[91,1] = PR[90,1] + -12.135;
   1:  PR[91,2] = PR[90,2] + -18.524;
   1:L PR[91] R[100]mm/sec CNT100;
   1:  PR[91,1] = PR[90,1] + -9.014;
   1:  PR[91,2] = PR[90,2] + -17.149;
   1:L PR[91] R[100]mm/sec CNT100;
   1:  PR[91,1] = PR[90,1] + -6.347;
   1:  PR[91,2] = PR[90,2] + -15.443;
   1:L PR[91] R[100]mm/sec CNT100;
   1:  PR[91,1] = PR[90,1] + -6.304;
   1:  PR[91,2] = PR[90,2] + -15.412;
   1:L PR[91] R[100]mm/sec CNT100;
   1:  PR[91,1] = PR[90,1] + -5.967;
   1:  PR[91,2] = PR[90,2] + -15.116;
   1:L PR[91] R[100]mm/sec CNT100;
   1:  PR[91,1] = PR[90,1] + -4.010;
   1:  PR[91,2] = PR[90,2] + -13.352;
   1:L PR[91] R[100]mm/sec CNT100;
   1:  PR[91,1] = PR[90,1] + -2.804;
   1:  PR[91,2] = PR[90,2] + -11.939;
   1:L PR[91] R[100]mm/sec CNT100;
   1:  PR[91,1] = PR[90,1] + -2.352;
   1:  PR[91,2] = PR[90,2] + -11.368;
   1:L PR[91] R[100]mm/sec CNT100;
   1:  PR[91,1] = PR[90,1] + -2.147;
   1:  PR[91,2] = PR[90,2] + -11.177;
   1:L PR[91] R[100]mm/sec CNT100;
   1:  PR[91,1] = PR[90,1] + -1.394;
   1:  PR[91,2] = PR[90,2] + -10.542;
   1:L PR[91] R[100]mm/sec CNT100;
   1:  PR[91,1] = PR[90,1] + -0.180;
   1:  PR[91,2] = PR[90,2] + -10.248;
   1:L PR[91] R[100]mm/sec CNT100;
   1:  PR[91,1] = PR[90,1] + 0.337;
   1:L PR[91] R[100]mm/sec CNT100;
   1:  PR[91,1] = PR[90,1] + 1.567;
   1:  PR[91,2] = PR[90,2] + -10.543;
   1:L PR[91] R[100]mm/sec CNT100;
   1:  PR[91,1] = PR[90,1] + 2.495;
   1:  PR[91,2] = PR[90,2] + -11.345;
   1:L PR[91] R[100]mm/sec CNT100;
   1:  PR[91,1] = PR[90,1] + 2.973;
   1:  PR[91,2] = PR[90,2] + -11.944;
   1:L PR[91] R[100]mm/sec CNT100;
   1:  PR[91,1] = PR[90,1] + 4.187;
   1:  PR[91,2] = PR[90,2] + -13.370;
   1:L PR[91] R[100]mm/sec CNT100;
   1:  PR[91,1] = PR[90,1] + 6.460;
   1:  PR[91,2] = PR[90,2] + -15.411;
   1:L PR[91] R[100]mm/sec CNT100;
   1:  PR[91,1] = PR[90,1] + 9.169;
   1:  PR[91,2] = PR[90,2] + -17.150;
   1:L PR[91] R[100]mm/sec CNT100;
   1:  PR[91,1] = PR[90,1] + 12.276;
   1:  PR[91,2] = PR[90,2] + -18.516;
   1:L PR[91] R[100]mm/sec CNT100;
   1:  PR[91,1] = PR[90,1] + 15.896;
   1:  PR[91,2] = PR[90,2] + -19.462;
   1:L PR[91] R[100]mm/sec CNT100;
   1:  PR[91,1] = PR[90,1] + 18.214;
   1:  PR[91,2] = PR[90,2] + -19.730;
   1:L PR[91] R[100]mm/sec CNT100;
   1:  PR[91,1] = PR[90,1] + 20.260;
   1:  PR[91,2] = PR[90,2] + -19.720;
   1:L PR[91] R[100]mm/sec CNT100;
   1:  PR[91,1] = PR[90,1] + 22.109;
   1:  PR[91,2] = PR[90,2] + -19.643;
   1:L PR[91] R[100]mm/sec CNT100;
   1:  PR[91,1] = PR[90,1] + 25.336;
   1:  PR[91,2] = PR[90,2] + -18.881;
   1:L PR[91] R[100]mm/sec CNT100;
   1:  PR[91,1] = PR[90,1] + 26.586;
   1:  PR[91,2] = PR[90,2] + -18.622;
   1:L PR[91] R[100]mm/sec CNT100;
   1:  PR[91,1] = PR[90,1] + 27.324;
   1:  PR[91,2] = PR[90,2] + -18.355;
   1:L PR[91] R[100]mm/sec CNT100;
   1:  PR[91,1] = PR[90,1] + 31.136;
   1:  PR[91,2] = PR[90,2] + -16.431;
   1:L PR[91] R[100]mm/sec CNT100;
   1:  PR[91,1] = PR[90,1] + 31.368;
   1:  PR[91,2] = PR[90,2] + -16.304;
   1:L PR[91] R[100]mm/sec CNT100;
   1:  PR[91,1] = PR[90,1] + 34.548;
   1:  PR[91,2] = PR[90,2] + -13.619;
   1:L PR[91] R[100]mm/sec CNT100;
   1:  PR[91,1] = PR[90,1] + 35.075;
   1:  PR[91,2] = PR[90,2] + -13.168;
   1:L PR[91] R[100]mm/sec CNT100;
   1:  PR[91,1] = PR[90,1] + 37.805;
   1:  PR[91,2] = PR[90,2] + -9.317;
   1:L PR[91] R[100]mm/sec CNT100;
   1:  PR[91,1] = PR[90,1] + 39.524;
   1:  PR[91,2] = PR[90,2] + -5.015;
   1:L PR[91] R[100]mm/sec CNT100;
   1:  PR[91,1] = PR[90,1] + 40.111;
   1:  PR[91,2] = PR[90,2] + -0.312;
   1:L PR[91] R[100]mm/sec CNT100;
   1:  PR[91,1] = PR[90,1] + 39.523;
   1:  PR[91,2] = PR[90,2] + 4.392;
   1:L PR[91] R[100]mm/sec CNT100;
   1:  PR[91,1] = PR[90,1] + 37.804;
   1:  PR[91,2] = PR[90,2] + 8.695;
   1:L PR[91] R[100]mm/sec CNT100;
   1:  PR[91,1] = PR[90,1] + 35.066;
   1:  PR[91,2] = PR[90,2] + 12.552;
   1:L PR[91] R[100]mm/sec CNT100;
   1:  PR[91,1] = PR[90,1] + 31.537;
   1:  PR[91,2] = PR[90,2] + 15.554;
   1:L PR[91] R[100]mm/sec CNT100;
   1:  PR[91,1] = PR[90,1] + 31.389;
   1:  PR[91,2] = PR[90,2] + 15.669;
   1:L PR[91] R[100]mm/sec CNT100;
   1:  PR[91,1] = PR[90,1] + 31.132;
   1:  PR[91,2] = PR[90,2] + 15.811;
   1:L PR[91] R[100]mm/sec CNT100;
   1:  PR[91,1] = PR[90,1] + 27.320;
   1:  PR[91,2] = PR[90,2] + 17.733;
   1:L PR[91] R[100]mm/sec CNT100;
   1:  PR[91,1] = PR[90,1] + 26.559;
   1:  PR[91,2] = PR[90,2] + 18.008;
   1:L PR[91] R[100]mm/sec CNT100;
   1:  PR[91,1] = PR[90,1] + 23.413;
   1:  PR[91,2] = PR[90,2] + 18.763;
   1:L PR[91] R[100]mm/sec CNT100;
   1:  PR[91,1] = PR[90,1] + 22.130;
   1:  PR[91,2] = PR[90,2] + 19.018;
   1:L PR[91] R[100]mm/sec CNT100;
   1:  PR[91,1] = PR[90,1] + 20.256;
   1:  PR[91,2] = PR[90,2] + 19.096;
   1:L PR[91] R[100]mm/sec CNT100;
   1:  PR[91,1] = PR[90,1] + 18.211;
   1:  PR[91,2] = PR[90,2] + 19.105;
   1:L PR[91] R[100]mm/sec CNT100;
   1:  PR[91,1] = PR[90,1] + 15.874;
   1:  PR[91,2] = PR[90,2] + 18.836;
   1:L PR[91] R[100]mm/sec CNT100;
   1:  PR[91,1] = PR[90,1] + 14.943;
   1:  PR[91,2] = PR[90,2] + 18.619;
   1:L PR[91] R[100]mm/sec CNT100;
   1:  PR[91,1] = PR[90,1] + 12.282;
   1:  PR[91,2] = PR[90,2] + 17.895;
   1:L PR[91] R[100]mm/sec CNT100;
   1:  PR[91,1] = PR[90,1] + 9.174;
   1:  PR[91,2] = PR[90,2] + 16.530;
   1:L PR[91] R[100]mm/sec CNT100;
   1:  PR[91,1] = PR[90,1] + 6.475;
   1:  PR[91,2] = PR[90,2] + 14.803;
   1:L PR[91] R[100]mm/sec CNT100;
   1:  PR[91,1] = PR[90,1] + 6.420;
   1:  PR[91,2] = PR[90,2] + 14.759;
   1:L PR[91] R[100]mm/sec CNT100;
   1:  PR[91,1] = PR[90,1] + 4.203;
   1:  PR[91,2] = PR[90,2] + 12.764;
   1:L PR[91] R[100]mm/sec CNT100;
   1:  PR[91,1] = PR[90,1] + 3.967;
   1:  PR[91,2] = PR[90,2] + 12.516;
   1:L PR[91] R[100]mm/sec CNT100;
   1:  PR[91,1] = PR[90,1] + 2.675;
   1:  PR[91,2] = PR[90,2] + 10.874;
   1:L PR[91] R[100]mm/sec CNT100;
   1:  PR[91,1] = PR[90,1] + 2.299;
   1:  PR[91,2] = PR[90,2] + 10.542;
   1:L PR[91] R[100]mm/sec CNT100;
   1:  PR[91,1] = PR[90,1] + 1.560;
   1:  PR[91,2] = PR[90,2] + 9.918;
   1:L PR[91] R[100]mm/sec CNT100;
   1:  PR[91,1] = PR[90,1] + 0.344;
   1:  PR[91,2] = PR[90,2] + 9.624;
   1:L PR[91] R[100]mm/sec CNT100;
   1:  PR[91,1] = PR[90,1] + -0.172;
   1:L PR[91] R[100]mm/sec CNT100;
   1:  PR[91] = PR[90];
   1:  PR[91,1] = PR[90,1] + -1.359;
   1:  PR[91,2] = PR[90,2] + 10.215;
   1:  PR[91,3] = PR[90,3] + 24.705;
   1:L PR[91] R[100]mm/sec CNT100;
   1:  PR[91,1] = PR[90,1] + -1.790;
   1:  PR[91,2] = PR[90,2] + 10.656;
   1:L PR[91] R[100]mm/sec CNT100;
   1:  PR[91,1] = PR[90,1] + -2.195;
   1:  PR[91,2] = PR[90,2] + 10.947;
   1:L PR[91] R[100]mm/sec CNT100;
   1:  PR[91,1] = PR[90,1] + -3.485;
   1:  PR[91,2] = PR[90,2] + 12.499;
   1:L PR[91] R[100]mm/sec CNT100;
   1:  PR[91,1] = PR[90,1] + -3.832;
   1:  PR[91,2] = PR[90,2] + 12.863;
   1:L PR[91] R[100]mm/sec CNT100;
   1:  PR[91,1] = PR[90,1] + -5.639;
   1:  PR[91,2] = PR[90,2] + 14.491;
   1:L PR[91] R[100]mm/sec CNT100;
   1:  PR[91,1] = PR[90,1] + -6.100;
   1:  PR[91,2] = PR[90,2] + 14.882;
   1:L PR[91] R[100]mm/sec CNT100;
   1:  PR[91,1] = PR[90,1] + -8.732;
   1:  PR[91,2] = PR[90,2] + 16.571;
   1:L PR[91] R[100]mm/sec CNT100;
   1:  PR[91,1] = PR[90,1] + -11.926;
   1:  PR[91,2] = PR[90,2] + 17.964;
   1:L PR[91] R[100]mm/sec CNT100;
   1:  PR[91,1] = PR[90,1] + -15.304;
   1:  PR[91,2] = PR[90,2] + 18.845;
   1:L PR[91] R[100]mm/sec CNT100;
   1:  PR[91,1] = PR[90,1] + -18.060;
   1:  PR[91,2] = PR[90,2] + 19.161;
   1:L PR[91] R[100]mm/sec CNT100;
   1:  PR[91,1] = PR[90,1] + -19.425;
   1:  PR[91,2] = PR[90,2] + 19.154;
   1:L PR[91] R[100]mm/sec CNT100;
   1:  PR[91,1] = PR[90,1] + -21.768;
   1:  PR[91,2] = PR[90,2] + 19.054;
   1:L PR[91] R[100]mm/sec CNT100;
   1:  PR[91,1] = PR[90,1] + -24.274;
   1:  PR[91,2] = PR[90,2] + 18.464;
   1:L PR[91] R[100]mm/sec CNT100;
   1:  PR[91,1] = PR[90,1] + -26.048;
   1:  PR[91,2] = PR[90,2] + 18.096;
   1:L PR[91] R[100]mm/sec CNT100;
   1:  PR[91,1] = PR[90,1] + -27.146;
   1:  PR[91,2] = PR[90,2] + 17.697;
   1:L PR[91] R[100]mm/sec CNT100;
   1:  PR[91,1] = PR[90,1] + -30.430;
   1:  PR[91,2] = PR[90,2] + 16.036;
   1:L PR[91] R[100]mm/sec CNT100;
   1:  PR[91,1] = PR[90,1] + -31.031;
   1:  PR[91,2] = PR[90,2] + 15.702;
   1:L PR[91] R[100]mm/sec CNT100;
   1:  PR[91,1] = PR[90,1] + -34.727;
   1:  PR[91,2] = PR[90,2] + 12.600;
   1:L PR[91] R[100]mm/sec CNT100;
   1:  PR[91,1] = PR[90,1] + -34.786;
   1:  PR[91,2] = PR[90,2] + 12.536;
   1:L PR[91] R[100]mm/sec CNT100;
   1:  PR[91,1] = PR[90,1] + -37.545;
   1:  PR[91,2] = PR[90,2] + 8.679;
   1:L PR[91] R[100]mm/sec CNT100;
   1:  PR[91,1] = PR[90,1] + -39.254;
   1:  PR[91,2] = PR[90,2] + 4.368;
   1:L PR[91] R[100]mm/sec CNT100;
   1:  PR[91,1] = PR[90,1] + -39.835;
   1:  PR[91,2] = PR[90,2] + -0.312;
   1:L PR[91] R[100]mm/sec CNT100;
   1:  PR[91,1] = PR[90,1] + -39.254;
   1:  PR[91,2] = PR[90,2] + -4.992;
   1:L PR[91] R[100]mm/sec CNT100;
   1:  PR[91,1] = PR[90,1] + -37.545;
   1:  PR[91,2] = PR[90,2] + -9.302;
   1:L PR[91] R[100]mm/sec CNT100;
   1:  PR[91,1] = PR[90,1] + -34.841;
   1:  PR[91,2] = PR[90,2] + -13.065;
   1:L PR[91] R[100]mm/sec CNT100;
   1:  PR[91,1] = PR[90,1] + -34.764;
   1:  PR[91,2] = PR[90,2] + -13.184;
   1:L PR[91] R[100]mm/sec CNT100;
   1:  PR[91,1] = PR[90,1] + -34.724;
   1:  PR[91,2] = PR[90,2] + -13.227;
   1:L PR[91] R[100]mm/sec CNT100;
   1:  PR[91,1] = PR[90,1] + -31.458;
   1:  PR[91,2] = PR[90,2] + -15.998;
   1:L PR[91] R[100]mm/sec CNT100;
   1:  PR[91,1] = PR[90,1] + -31.053;
   1:  PR[91,2] = PR[90,2] + -16.314;
   1:L PR[91] R[100]mm/sec CNT100;
   1:  PR[91,1] = PR[90,1] + -30.430;
   1:  PR[91,2] = PR[90,2] + -16.660;
   1:L PR[91] R[100]mm/sec CNT100;
   1:  PR[91,1] = PR[90,1] + -27.146;
   1:  PR[91,2] = PR[90,2] + -18.321;
   1:L PR[91] R[100]mm/sec CNT100;
   1:  PR[91,1] = PR[90,1] + -26.027;
   1:  PR[91,2] = PR[90,2] + -18.727;
   1:L PR[91] R[100]mm/sec CNT100;
   1:  PR[91,1] = PR[90,1] + -23.416;
   1:  PR[91,2] = PR[90,2] + -19.354;
   1:L PR[91] R[100]mm/sec CNT100;
   1:  PR[91,1] = PR[90,1] + -21.793;
   1:  PR[91,2] = PR[90,2] + -19.677;
   1:L PR[91] R[100]mm/sec CNT100;
   1:  PR[91,1] = PR[90,1] + -19.425;
   1:  PR[91,2] = PR[90,2] + -19.778;
   1:L PR[91] R[100]mm/sec CNT100;
   1:  PR[91,1] = PR[90,1] + -18.060;
   1:  PR[91,2] = PR[90,2] + -19.785;
   1:L PR[91] R[100]mm/sec CNT100;
   1:  PR[91,1] = PR[90,1] + -15.285;
   1:  PR[91,2] = PR[90,2] + -19.467;
   1:L PR[91] R[100]mm/sec CNT100;
   1:  PR[91,1] = PR[90,1] + -14.952;
   1:  PR[91,2] = PR[90,2] + -19.389;
   1:L PR[91] R[100]mm/sec CNT100;
   1:  PR[91,1] = PR[90,1] + -11.927;
   1:  PR[91,2] = PR[90,2] + -18.589;
   1:L PR[91] R[100]mm/sec CNT100;
   1:  PR[91,1] = PR[90,1] + -8.719;
   1:  PR[91,2] = PR[90,2] + -17.187;
   1:L PR[91] R[100]mm/sec CNT100;
   1:  PR[91,1] = PR[90,1] + -6.162;
   1:  PR[91,2] = PR[90,2] + -15.551;
   1:L PR[91] R[100]mm/sec CNT100;
   1:  PR[91,1] = PR[90,1] + -6.060;
   1:  PR[91,2] = PR[90,2] + -15.478;
   1:L PR[91] R[100]mm/sec CNT100;
   1:  PR[91,1] = PR[90,1] + -5.543;
   1:  PR[91,2] = PR[90,2] + -15.025;
   1:L PR[91] R[100]mm/sec CNT100;
   1:  PR[91,1] = PR[90,1] + -3.804;
   1:  PR[91,2] = PR[90,2] + -13.457;
   1:L PR[91] R[100]mm/sec CNT100;
   1:  PR[91,1] = PR[90,1] + -2.184;
   1:  PR[91,2] = PR[90,2] + -11.558;
   1:L PR[91] R[100]mm/sec CNT100;
   1:  PR[91,1] = PR[90,1] + -1.791;
   1:  PR[91,2] = PR[90,2] + -11.279;
   1:L PR[91] R[100]mm/sec CNT100;
   1:  PR[91,1] = PR[90,1] + -1.366;
   1:  PR[91,2] = PR[90,2] + -10.842;
   1:L PR[91] R[100]mm/sec CNT100;
   1:  PR[91,1] = PR[90,1] + 0.063;
   1:  PR[91,2] = PR[90,2] + -10.500;
   1:L PR[91] R[100]mm/sec CNT100;
   1:  PR[91,1] = PR[90,1] + 1.521;
   1:  PR[91,2] = PR[90,2] + -10.835;
   1:L PR[91] R[100]mm/sec CNT100;
   1:  PR[91,1] = PR[90,1] + 1.954;
   1:  PR[91,2] = PR[90,2] + -11.277;
   1:L PR[91] R[100]mm/sec CNT100;
   1:  PR[91,1] = PR[90,1] + 2.351;
   1:  PR[91,2] = PR[90,2] + -11.559;
   1:L PR[91] R[100]mm/sec CNT100;
   1:  PR[91,1] = PR[90,1] + 3.978;
   1:  PR[91,2] = PR[90,2] + -13.472;
   1:L PR[91] R[100]mm/sec CNT100;
   1:  PR[91,1] = PR[90,1] + 6.215;
   1:  PR[91,2] = PR[90,2] + -15.475;
   1:L PR[91] R[100]mm/sec CNT100;
   1:  PR[91,1] = PR[90,1] + 8.875;
   1:  PR[91,2] = PR[90,2] + -17.188;
   1:L PR[91] R[100]mm/sec CNT100;
   1:  PR[91,1] = PR[90,1] + 12.073;
   1:  PR[91,2] = PR[90,2] + -18.583;
   1:L PR[91] R[100]mm/sec CNT100;
   1:  PR[91,1] = PR[90,1] + 15.459;
   1:  PR[91,2] = PR[90,2] + -19.468;
   1:L PR[91] R[100]mm/sec CNT100;
   1:  PR[91,1] = PR[90,1] + 18.209;
   1:  PR[91,2] = PR[90,2] + -19.785;
   1:L PR[91] R[100]mm/sec CNT100;
   1:  PR[91,1] = PR[90,1] + 19.573;
   1:  PR[91,2] = PR[90,2] + -19.778;
   1:L PR[91] R[100]mm/sec CNT100;
   1:  PR[91,1] = PR[90,1] + 21.910;
   1:  PR[91,2] = PR[90,2] + -19.681;
   1:L PR[91] R[100]mm/sec CNT100;
   1:  PR[91,1] = PR[90,1] + 24.414;
   1:  PR[91,2] = PR[90,2] + -19.090;
   1:L PR[91] R[100]mm/sec CNT100;
   1:  PR[91,1] = PR[90,1] + 26.193;
   1:  PR[91,2] = PR[90,2] + -18.721;
   1:L PR[91] R[100]mm/sec CNT100;
   1:  PR[91,1] = PR[90,1] + 27.297;
   1:  PR[91,2] = PR[90,2] + -18.322;
   1:L PR[91] R[100]mm/sec CNT100;
   1:  PR[91,1] = PR[90,1] + 30.583;
   1:  PR[91,2] = PR[90,2] + -16.664;
   1:L PR[91] R[100]mm/sec CNT100;
   1:  PR[91,1] = PR[90,1] + 31.180;
   1:  PR[91,2] = PR[90,2] + -16.334;
   1:L PR[91] R[100]mm/sec CNT100;
   1:  PR[91,1] = PR[90,1] + 34.695;
   1:  PR[91,2] = PR[90,2] + -13.367;
   1:L PR[91] R[100]mm/sec CNT100;
   1:  PR[91,1] = PR[90,1] + 34.895;
   1:  PR[91,2] = PR[90,2] + -13.209;
   1:L PR[91] R[100]mm/sec CNT100;
   1:  PR[91,1] = PR[90,1] + 34.940;
   1:  PR[91,2] = PR[90,2] + -13.160;
   1:L PR[91] R[100]mm/sec CNT100;
   1:  PR[91,1] = PR[90,1] + 37.702;
   1:  PR[91,2] = PR[90,2] + -9.296;
   1:L PR[91] R[100]mm/sec CNT100;
   1:  PR[91,1] = PR[90,1] + 39.410;
   1:  PR[91,2] = PR[90,2] + -5.009;
   1:L PR[91] R[100]mm/sec CNT100;
   1:  PR[91,1] = PR[90,1] + 39.992;
   1:  PR[91,2] = PR[90,2] + -0.312;
   1:L PR[91] R[100]mm/sec CNT100;
   1:  PR[91,1] = PR[90,1] + 39.410;
   1:  PR[91,2] = PR[90,2] + 4.386;
   1:L PR[91] R[100]mm/sec CNT100;
   1:  PR[91,1] = PR[90,1] + 37.701;
   1:  PR[91,2] = PR[90,2] + 8.675;
   1:L PR[91] R[100]mm/sec CNT100;
   1:  PR[91,1] = PR[90,1] + 34.937;
   1:  PR[91,2] = PR[90,2] + 12.539;
   1:L PR[91] R[100]mm/sec CNT100;
   1:  PR[91,1] = PR[90,1] + 34.874;
   1:  PR[91,2] = PR[90,2] + 12.607;
   1:L PR[91] R[100]mm/sec CNT100;
   1:  PR[91,1] = PR[90,1] + 31.603;
   1:  PR[91,2] = PR[90,2] + 15.387;
   1:L PR[91] R[100]mm/sec CNT100;
   1:  PR[91,1] = PR[90,1] + 31.202;
   1:  PR[91,2] = PR[90,2] + 15.699;
   1:L PR[91] R[100]mm/sec CNT100;
   1:  PR[91,1] = PR[90,1] + 30.579;
   1:  PR[91,2] = PR[90,2] + 16.042;
   1:L PR[91] R[100]mm/sec CNT100;
   1:  PR[91,1] = PR[90,1] + 27.292;
   1:  PR[91,2] = PR[90,2] + 17.700;
   1:L PR[91] R[100]mm/sec CNT100;
   1:  PR[91,1] = PR[90,1] + 26.168;
   1:  PR[91,2] = PR[90,2] + 18.106;
   1:L PR[91] R[100]mm/sec CNT100;
   1:  PR[91,1] = PR[90,1] + 23.557;
   1:  PR[91,2] = PR[90,2] + 18.733;
   1:L PR[91] R[100]mm/sec CNT100;
   1:  PR[91,1] = PR[90,1] + 21.932;
   1:  PR[91,2] = PR[90,2] + 19.056;
   1:L PR[91] R[100]mm/sec CNT100;
   1:  PR[91,1] = PR[90,1] + 19.571;
   1:  PR[91,2] = PR[90,2] + 19.155;
   1:L PR[91] R[100]mm/sec CNT100;
   1:  PR[91,1] = PR[90,1] + 18.207;
   1:  PR[91,2] = PR[90,2] + 19.161;
   1:L PR[91] R[100]mm/sec CNT100;
   1:  PR[91,1] = PR[90,1] + 15.439;
   1:  PR[91,2] = PR[90,2] + 18.842;
   1:L PR[91] R[100]mm/sec CNT100;
   1:  PR[91,1] = PR[90,1] + 15.107;
   1:  PR[91,2] = PR[90,2] + 18.764;
   1:L PR[91] R[100]mm/sec CNT100;
   1:  PR[91,1] = PR[90,1] + 12.076;
   1:  PR[91,2] = PR[90,2] + 17.960;
   1:L PR[91] R[100]mm/sec CNT100;
   1:  PR[91,1] = PR[90,1] + 8.884;
   1:  PR[91,2] = PR[90,2] + 16.571;
   1:L PR[91] R[100]mm/sec CNT100;
   1:  PR[91,1] = PR[90,1] + 6.255;
   1:  PR[91,2] = PR[90,2] + 14.886;
   1:L PR[91] R[100]mm/sec CNT100;
   1:  PR[91,1] = PR[90,1] + 6.132;
   1:  PR[91,2] = PR[90,2] + 14.789;
   1:L PR[91] R[100]mm/sec CNT100;
   1:  PR[91,1] = PR[90,1] + 4.009;
   1:  PR[91,2] = PR[90,2] + 12.880;
   1:L PR[91] R[100]mm/sec CNT100;
   1:  PR[91,1] = PR[90,1] + 3.674;
   1:  PR[91,2] = PR[90,2] + 12.528;
   1:L PR[91] R[100]mm/sec CNT100;
   1:  PR[91,1] = PR[90,1] + 2.611;
   1:  PR[91,2] = PR[90,2] + 11.177;
   1:L PR[91] R[100]mm/sec CNT100;
   1:  PR[91,1] = PR[90,1] + 2.255;
   1:  PR[91,2] = PR[90,2] + 10.866;
   1:L PR[91] R[100]mm/sec CNT100;
   1:  PR[91,1] = PR[90,1] + 1.957;
   1:  PR[91,2] = PR[90,2] + 10.655;
   1:L PR[91] R[100]mm/sec CNT100;
   1:  PR[91,1] = PR[90,1] + 1.528;
   1:  PR[91,2] = PR[90,2] + 10.214;
   1:L PR[91] R[100]mm/sec CNT100;
   1:  PR[91,1] = PR[90,1] + 0.065;
   1:  PR[91,2] = PR[90,2] + 9.875;
   1:L PR[91] R[100]mm/sec CNT100;
   1:  PR[91] = PR[90];
   1:  PR[91,1] = PR[90,1] + -1.263;
   1:  PR[91,2] = PR[90,2] + 10.569;
   1:  PR[91,3] = PR[90,3] + 25.315;
   1:L PR[91] R[100]mm/sec CNT100;
   1:  PR[91,1] = PR[90,1] + -1.470;
   1:  PR[91,2] = PR[90,2] + 10.780;
   1:L PR[91] R[100]mm/sec CNT100;
   1:  PR[91,1] = PR[90,1] + -2.176;
   1:  PR[91,2] = PR[90,2] + 11.289;
   1:L PR[91] R[100]mm/sec CNT100;
   1:  PR[91,1] = PR[90,1] + -3.194;
   1:  PR[91,2] = PR[90,2] + 12.514;
   1:L PR[91] R[100]mm/sec CNT100;
   1:  PR[91,1] = PR[90,1] + -3.640;
   1:  PR[91,2] = PR[90,2] + 12.981;
   1:L PR[91] R[100]mm/sec CNT100;
   1:  PR[91,1] = PR[90,1] + -5.259;
   1:  PR[91,2] = PR[90,2] + 14.440;
   1:L PR[91] R[100]mm/sec CNT100;
   1:  PR[91,1] = PR[90,1] + -5.666;
   1:  PR[91,2] = PR[90,2] + 14.799;
   1:L PR[91] R[100]mm/sec CNT100;
   1:  PR[91,1] = PR[90,1] + -5.860;
   1:  PR[91,2] = PR[90,2] + 14.952;
   1:L PR[91] R[100]mm/sec CNT100;
   1:  PR[91,1] = PR[90,1] + -8.444;
   1:  PR[91,2] = PR[90,2] + 16.613;
   1:L PR[91] R[100]mm/sec CNT100;
   1:  PR[91,1] = PR[90,1] + -11.728;
   1:  PR[91,2] = PR[90,2] + 18.042;
   1:L PR[91] R[100]mm/sec CNT100;
   1:  PR[91,1] = PR[90,1] + -14.896;
   1:  PR[91,2] = PR[90,2] + 18.861;
   1:L PR[91] R[100]mm/sec CNT100;
   1:  PR[91,1] = PR[90,1] + -18.054;
   1:  PR[91,2] = PR[90,2] + 19.216;
   1:L PR[91] R[100]mm/sec CNT100;
   1:  PR[91,1] = PR[90,1] + -18.740;
   1:  PR[91,2] = PR[90,2] + 19.213;
   1:L PR[91] R[100]mm/sec CNT100;
   1:  PR[91,1] = PR[90,1] + -21.571;
   1:  PR[91,2] = PR[90,2] + 19.092;
   1:L PR[91] R[100]mm/sec CNT100;
   1:  PR[91,1] = PR[90,1] + -23.357;
   1:  PR[91,2] = PR[90,2] + 18.672;
   1:L PR[91] R[100]mm/sec CNT100;
   1:  PR[91,1] = PR[90,1] + -25.659;
   1:  PR[91,2] = PR[90,2] + 18.194;
   1:L PR[91] R[100]mm/sec CNT100;
   1:  PR[91,1] = PR[90,1] + -27.120;
   1:  PR[91,2] = PR[90,2] + 17.663;
   1:L PR[91] R[100]mm/sec CNT100;
   1:  PR[91,1] = PR[90,1] + -29.880;
   1:  PR[91,2] = PR[90,2] + 16.267;
   1:L PR[91] R[100]mm/sec CNT100;
   1:  PR[91,1] = PR[90,1] + -30.846;
   1:  PR[91,2] = PR[90,2] + 15.732;
   1:L PR[91] R[100]mm/sec CNT100;
   1:  PR[91,1] = PR[90,1] + -33.892;
   1:  PR[91,2] = PR[90,2] + 13.164;
   1:L PR[91] R[100]mm/sec CNT100;
   1:  PR[91,1] = PR[90,1] + -34.433;
   1:  PR[91,2] = PR[90,2] + 12.735;
   1:L PR[91] R[100]mm/sec CNT100;
   1:  PR[91,1] = PR[90,1] + -34.711;
   1:  PR[91,2] = PR[90,2] + 12.436;
   1:L PR[91] R[100]mm/sec CNT100;
   1:  PR[91,1] = PR[90,1] + -37.299;
   1:  PR[91,2] = PR[90,2] + 8.823;
   1:L PR[91] R[100]mm/sec CNT100;
   1:  PR[91,1] = PR[90,1] + -37.386;
   1:  PR[91,2] = PR[90,2] + 8.692;
   1:L PR[91] R[100]mm/sec CNT100;
   1:  PR[91,1] = PR[90,1] + -37.436;
   1:  PR[91,2] = PR[90,2] + 8.578;
   1:L PR[91] R[100]mm/sec CNT100;
   1:  PR[91,1] = PR[90,1] + -39.135;
   1:  PR[91,2] = PR[90,2] + 4.322;
   1:L PR[91] R[100]mm/sec CNT100;
   1:  PR[91,1] = PR[90,1] + -39.716;
   1:  PR[91,2] = PR[90,2] + -0.312;
   1:L PR[91] R[100]mm/sec CNT100;
   1:  PR[91,1] = PR[90,1] + -39.130;
   1:  PR[91,2] = PR[90,2] + -4.982;
   1:L PR[91] R[100]mm/sec CNT100;
   1:  PR[91,1] = PR[90,1] + -37.383;
   1:  PR[91,2] = PR[90,2] + -9.308;
   1:L PR[91] R[100]mm/sec CNT100;
   1:  PR[91,1] = PR[90,1] + -34.928;
   1:  PR[91,2] = PR[90,2] + -12.716;
   1:L PR[91] R[100]mm/sec CNT100;
   1:  PR[91,1] = PR[90,1] + -34.688;
   1:  PR[91,2] = PR[90,2] + -13.085;
   1:L PR[91] R[100]mm/sec CNT100;
   1:  PR[91,1] = PR[90,1] + -34.416;
   1:  PR[91,2] = PR[90,2] + -13.377;
   1:L PR[91] R[100]mm/sec CNT100;
   1:  PR[91,1] = PR[90,1] + -31.527;
   1:  PR[91,2] = PR[90,2] + -15.828;
   1:L PR[91] R[100]mm/sec CNT100;
   1:  PR[91,1] = PR[90,1] + -30.869;
   1:  PR[91,2] = PR[90,2] + -16.343;
   1:L PR[91] R[100]mm/sec CNT100;
   1:  PR[91,1] = PR[90,1] + -29.880;
   1:  PR[91,2] = PR[90,2] + -16.891;
   1:L PR[91] R[100]mm/sec CNT100;
   1:  PR[91,1] = PR[90,1] + -27.120;
   1:  PR[91,2] = PR[90,2] + -18.287;
   1:L PR[91] R[100]mm/sec CNT100;
   1:  PR[91,1] = PR[90,1] + -25.638;
   1:  PR[91,2] = PR[90,2] + -18.825;
   1:L PR[91] R[100]mm/sec CNT100;
   1:  PR[91,1] = PR[90,1] + -23.563;
   1:  PR[91,2] = PR[90,2] + -19.323;
   1:L PR[91] R[100]mm/sec CNT100;
   1:  PR[91,1] = PR[90,1] + -21.596;
   1:  PR[91,2] = PR[90,2] + -19.715;
   1:L PR[91] R[100]mm/sec CNT100;
   1:  PR[91,1] = PR[90,1] + -18.740;
   1:  PR[91,2] = PR[90,2] + -19.837;
   1:L PR[91] R[100]mm/sec CNT100;
   1:  PR[91,1] = PR[90,1] + -18.054;
   1:  PR[91,2] = PR[90,2] + -19.840;
   1:L PR[91] R[100]mm/sec CNT100;
   1:  PR[91,1] = PR[90,1] + -14.896;
   1:  PR[91,2] = PR[90,2] + -19.485;
   1:L PR[91] R[100]mm/sec CNT100;
   1:  PR[91,1] = PR[90,1] + -11.725;
   1:  PR[91,2] = PR[90,2] + -18.665;
   1:L PR[91] R[100]mm/sec CNT100;
   1:  PR[91,1] = PR[90,1] + -8.426;
   1:  PR[91,2] = PR[90,2] + -17.226;
   1:L PR[91] R[100]mm/sec CNT100;
   1:  PR[91,1] = PR[90,1] + -5.977;
   1:  PR[91,2] = PR[90,2] + -15.660;
   1:L PR[91] R[100]mm/sec CNT100;
   1:  PR[91,1] = PR[90,1] + -5.816;
   1:  PR[91,2] = PR[90,2] + -15.543;
   1:L PR[91] R[100]mm/sec CNT100;
   1:  PR[91,1] = PR[90,1] + -5.119;
   1:  PR[91,2] = PR[90,2] + -14.933;
   1:L PR[91] R[100]mm/sec CNT100;
   1:  PR[91,1] = PR[90,1] + -3.597;
   1:  PR[91,2] = PR[90,2] + -13.562;
   1:L PR[91] R[100]mm/sec CNT100;
   1:  PR[91,1] = PR[90,1] + -2.167;
   1:  PR[91,2] = PR[90,2] + -11.885;
   1:L PR[91] R[100]mm/sec CNT100;
   1:  PR[91,1] = PR[90,1] + -0.604;
   1:  PR[91,2] = PR[90,2] + -10.766;
   1:L PR[91] R[100]mm/sec CNT100;
   1:  PR[91,1] = PR[90,1] + -0.055;
   1:  PR[91,2] = PR[90,2] + -10.961;
   1:L PR[91] R[100]mm/sec CNT100;
   1:  PR[91,1] = PR[90,1] + 1.044;
   1:L PR[91] R[100]mm/sec CNT100;
   1:  PR[91,1] = PR[90,1] + 2.334;
   1:  PR[91,2] = PR[90,2] + -11.886;
   1:L PR[91] R[100]mm/sec CNT100;
   1:  PR[91,1] = PR[90,1] + 3.770;
   1:  PR[91,2] = PR[90,2] + -13.575;
   1:L PR[91] R[100]mm/sec CNT100;
   1:  PR[91,1] = PR[90,1] + 5.967;
   1:  PR[91,2] = PR[90,2] + -15.538;
   1:L PR[91] R[100]mm/sec CNT100;
   1:  PR[91,1] = PR[90,1] + 8.386;
   1:  PR[91,2] = PR[90,2] + -17.087;
   1:L PR[91] R[100]mm/sec CNT100;
   1:  PR[91,1] = PR[90,1] + 8.602;
   1:  PR[91,2] = PR[90,2] + -17.236;
   1:L PR[91] R[100]mm/sec CNT100;
   1:  PR[91,1] = PR[90,1] + 11.873;
   1:  PR[91,2] = PR[90,2] + -18.660;
   1:L PR[91] R[100]mm/sec CNT100;
   1:  PR[91,1] = PR[90,1] + 15.050;
   1:  PR[91,2] = PR[90,2] + -19.484;
   1:L PR[91] R[100]mm/sec CNT100;
   1:  PR[91,1] = PR[90,1] + 18.203;
   1:  PR[91,2] = PR[90,2] + -19.840;
   1:L PR[91] R[100]mm/sec CNT100;
   1:  PR[91,1] = PR[90,1] + 18.886;
   1:  PR[91,2] = PR[90,2] + -19.837;
   1:L PR[91] R[100]mm/sec CNT100;
   1:  PR[91,1] = PR[90,1] + 21.710;
   1:  PR[91,2] = PR[90,2] + -19.719;
   1:L PR[91] R[100]mm/sec CNT100;
   1:  PR[91,1] = PR[90,1] + 23.492;
   1:  PR[91,2] = PR[90,2] + -19.298;
   1:L PR[91] R[100]mm/sec CNT100;
   1:  PR[91,1] = PR[90,1] + 25.801;
   1:  PR[91,2] = PR[90,2] + -18.820;
   1:L PR[91] R[100]mm/sec CNT100;
   1:  PR[91,1] = PR[90,1] + 27.269;
   1:  PR[91,2] = PR[90,2] + -18.289;
   1:L PR[91] R[100]mm/sec CNT100;
   1:  PR[91,1] = PR[90,1] + 30.029;
   1:  PR[91,2] = PR[90,2] + -16.896;
   1:L PR[91] R[100]mm/sec CNT100;
   1:  PR[91,1] = PR[90,1] + 30.993;
   1:  PR[91,2] = PR[90,2] + -16.365;
   1:L PR[91] R[100]mm/sec CNT100;
   1:  PR[91,1] = PR[90,1] + 34.041;
   1:  PR[91,2] = PR[90,2] + -13.791;
   1:L PR[91] R[100]mm/sec CNT100;
   1:  PR[91,1] = PR[90,1] + 34.581;
   1:  PR[91,2] = PR[90,2] + -13.365;
   1:L PR[91] R[100]mm/sec CNT100;
   1:  PR[91,1] = PR[90,1] + 34.861;
   1:  PR[91,2] = PR[90,2] + -13.065;
   1:L PR[91] R[100]mm/sec CNT100;
   1:  PR[91,1] = PR[90,1] + 37.453;
   1:  PR[91,2] = PR[90,2] + -9.445;
   1:L PR[91] R[100]mm/sec CNT100;
   1:  PR[91,1] = PR[90,1] + 37.544;
   1:  PR[91,2] = PR[90,2] + -9.307;
   1:L PR[91] R[100]mm/sec CNT100;
   1:  PR[91,1] = PR[90,1] + 37.593;
   1:  PR[91,2] = PR[90,2] + -9.198;
   1:L PR[91] R[100]mm/sec CNT100;
   1:  PR[91,1] = PR[90,1] + 39.291;
   1:  PR[91,2] = PR[90,2] + -4.965;
   1:L PR[91] R[100]mm/sec CNT100;
   1:  PR[91,1] = PR[90,1] + 39.872;
   1:  PR[91,2] = PR[90,2] + -0.313;
   1:L PR[91] R[100]mm/sec CNT100;
   1:  PR[91,1] = PR[90,1] + 39.272;
   1:  PR[91,2] = PR[90,2] + 4.413;
   1:L PR[91] R[100]mm/sec CNT100;
   1:  PR[91,1] = PR[90,1] + 37.593;
   1:  PR[91,2] = PR[90,2] + 8.574;
   1:L PR[91] R[100]mm/sec CNT100;
   1:  PR[91,1] = PR[90,1] + 37.554;
   1:  PR[91,2] = PR[90,2] + 8.659;
   1:L PR[91] R[100]mm/sec CNT100;
   1:  PR[91,1] = PR[90,1] + 35.081;
   1:  PR[91,2] = PR[90,2] + 12.094;
   1:L PR[91] R[100]mm/sec CNT100;
   1:  PR[91,1] = PR[90,1] + 34.838;
   1:  PR[91,2] = PR[90,2] + 12.465;
   1:L PR[91] R[100]mm/sec CNT100;
   1:  PR[91,1] = PR[90,1] + 34.561;
   1:  PR[91,2] = PR[90,2] + 12.763;
   1:L PR[91] R[100]mm/sec CNT100;
   1:  PR[91,1] = PR[90,1] + 31.669;
   1:  PR[91,2] = PR[90,2] + 15.221;
   1:L PR[91] R[100]mm/sec CNT100;
   1:  PR[91,1] = PR[90,1] + 31.015;
   1:  PR[91,2] = PR[90,2] + 15.729;
   1:L PR[91] R[100]mm/sec CNT100;
   1:  PR[91,1] = PR[90,1] + 30.026;
   1:  PR[91,2] = PR[90,2] + 16.275;
   1:L PR[91] R[100]mm/sec CNT100;
   1:  PR[91,1] = PR[90,1] + 27.265;
   1:  PR[91,2] = PR[90,2] + 17.667;
   1:L PR[91] R[100]mm/sec CNT100;
   1:  PR[91,1] = PR[90,1] + 25.776;
   1:  PR[91,2] = PR[90,2] + 18.205;
   1:L PR[91] R[100]mm/sec CNT100;
   1:  PR[91,1] = PR[90,1] + 23.702;
   1:  PR[91,2] = PR[90,2] + 18.703;
   1:L PR[91] R[100]mm/sec CNT100;
   1:  PR[91,1] = PR[90,1] + 21.733;
   1:  PR[91,2] = PR[90,2] + 19.094;
   1:L PR[91] R[100]mm/sec CNT100;
   1:  PR[91,1] = PR[90,1] + 18.885;
   1:  PR[91,2] = PR[90,2] + 19.213;
   1:L PR[91] R[100]mm/sec CNT100;
   1:  PR[91,1] = PR[90,1] + 18.202;
   1:  PR[91,2] = PR[90,2] + 19.216;
   1:L PR[91] R[100]mm/sec CNT100;
   1:  PR[91,1] = PR[90,1] + 15.050;
   1:  PR[91,2] = PR[90,2] + 18.860;
   1:L PR[91] R[100]mm/sec CNT100;
   1:  PR[91,1] = PR[90,1] + 11.876;
   1:  PR[91,2] = PR[90,2] + 18.037;
   1:L PR[91] R[100]mm/sec CNT100;
   1:  PR[91,1] = PR[90,1] + 8.595;
   1:  PR[91,2] = PR[90,2] + 16.613;
   1:L PR[91] R[100]mm/sec CNT100;
   1:  PR[91,1] = PR[90,1] + 6.180;
   1:  PR[91,2] = PR[90,2] + 15.071;
   1:L PR[91] R[100]mm/sec CNT100;
   1:  PR[91,1] = PR[90,1] + 5.832;
   1:  PR[91,2] = PR[90,2] + 14.808;
   1:L PR[91] R[100]mm/sec CNT100;
   1:  PR[91,1] = PR[90,1] + 3.815;
   1:  PR[91,2] = PR[90,2] + 12.996;
   1:L PR[91] R[100]mm/sec CNT100;
   1:  PR[91,1] = PR[90,1] + 3.381;
   1:  PR[91,2] = PR[90,2] + 12.540;
   1:L PR[91] R[100]mm/sec CNT100;
   1:  PR[91,1] = PR[90,1] + 2.544;
   1:  PR[91,2] = PR[90,2] + 11.477;
   1:L PR[91] R[100]mm/sec CNT100;
   1:  PR[91,1] = PR[90,1] + 2.406;
   1:  PR[91,2] = PR[90,2] + 11.358;
   1:L PR[91] R[100]mm/sec CNT100;
   1:  PR[91,1] = PR[90,1] + 2.316;
   1:  PR[91,2] = PR[90,2] + 11.240;
   1:L PR[91] R[100]mm/sec CNT100;
   1:  PR[91,1] = PR[90,1] + 0.985;
   1:  PR[91,2] = PR[90,2] + 10.311;
   1:L PR[91] R[100]mm/sec CNT100;
   1:  PR[91,1] = PR[90,1] + -0.684;
   1:  PR[91,2] = PR[90,2] + 10.310;
   1:L PR[91] R[100]mm/sec CNT100;
   1:  PR[91] = PR[90];
   1:  PR[91,1] = PR[90,1] + -1.384;
   1:  PR[91,2] = PR[90,2] + 10.948;
   1:  PR[91,3] = PR[90,3] + 25.925;
   1:L PR[91] R[100]mm/sec CNT100;
   1:  PR[91,1] = PR[90,1] + -1.590;
   1:  PR[91,2] = PR[90,2] + 11.216;
   1:L PR[91] R[100]mm/sec CNT100;
   1:  PR[91,1] = PR[90,1] + -1.619;
   1:  PR[91,2] = PR[90,2] + 11.244;
   1:L PR[91] R[100]mm/sec CNT100;
   1:  PR[91,1] = PR[90,1] + -2.157;
   1:  PR[91,2] = PR[90,2] + 11.632;
   1:L PR[91] R[100]mm/sec CNT100;
   1:  PR[91,1] = PR[90,1] + -2.903;
   1:  PR[91,2] = PR[90,2] + 12.528;
   1:L PR[91] R[100]mm/sec CNT100;
   1:  PR[91,1] = PR[90,1] + -3.447;
   1:  PR[91,2] = PR[90,2] + 13.098;
   1:L PR[91] R[100]mm/sec CNT100;
   1:  PR[91,1] = PR[90,1] + -5.383;
   1:  PR[91,2] = PR[90,2] + 14.834;
   1:L PR[91] R[100]mm/sec CNT100;
   1:  PR[91,1] = PR[90,1] + -5.640;
   1:  PR[91,2] = PR[90,2] + 15.037;
   1:L PR[91] R[100]mm/sec CNT100;
   1:  PR[91,1] = PR[90,1] + -8.157;
   1:  PR[91,2] = PR[90,2] + 16.656;
   1:L PR[91] R[100]mm/sec CNT100;
   1:  PR[91,1] = PR[90,1] + -11.531;
   1:  PR[91,2] = PR[90,2] + 18.121;
   1:L PR[91] R[100]mm/sec CNT100;
   1:  PR[91,1] = PR[90,1] + -14.566;
   1:  PR[91,2] = PR[90,2] + 18.905;
   1:L PR[91] R[100]mm/sec CNT100;
   1:  PR[91,1] = PR[90,1] + -18.019;
   1:  PR[91,2] = PR[90,2] + 19.269;
   1:L PR[91] R[100]mm/sec CNT100;
   1:  PR[91,1] = PR[90,1] + -21.375;
   1:  PR[91,2] = PR[90,2] + 19.130;
   1:L PR[91] R[100]mm/sec CNT100;
   1:  PR[91,1] = PR[90,1] + -22.439;
   1:  PR[91,2] = PR[90,2] + 18.879;
   1:L PR[91] R[100]mm/sec CNT100;
   1:  PR[91,1] = PR[90,1] + -25.270;
   1:  PR[91,2] = PR[90,2] + 18.292;
   1:L PR[91] R[100]mm/sec CNT100;
   1:  PR[91,1] = PR[90,1] + -27.094;
   1:  PR[91,2] = PR[90,2] + 17.629;
   1:L PR[91] R[100]mm/sec CNT100;
   1:  PR[91,1] = PR[90,1] + -29.329;
   1:  PR[91,2] = PR[90,2] + 16.499;
   1:L PR[91] R[100]mm/sec CNT100;
   1:  PR[91,1] = PR[90,1] + -30.661;
   1:  PR[91,2] = PR[90,2] + 15.760;
   1:L PR[91] R[100]mm/sec CNT100;
   1:  PR[91,1] = PR[90,1] + -33.242;
   1:  PR[91,2] = PR[90,2] + 13.584;
   1:L PR[91] R[100]mm/sec CNT100;
   1:  PR[91,1] = PR[90,1] + -34.125;
   1:  PR[91,2] = PR[90,2] + 12.886;
   1:L PR[91] R[100]mm/sec CNT100;
   1:  PR[91,1] = PR[90,1] + -34.635;
   1:  PR[91,2] = PR[90,2] + 12.337;
   1:L PR[91] R[100]mm/sec CNT100;
   1:  PR[91,1] = PR[90,1] + -36.923;
   1:  PR[91,2] = PR[90,2] + 9.143;
   1:L PR[91] R[100]mm/sec CNT100;
   1:  PR[91,1] = PR[90,1] + -37.208;
   1:  PR[91,2] = PR[90,2] + 8.709;
   1:L PR[91] R[100]mm/sec CNT100;
   1:  PR[91,1] = PR[90,1] + -37.391;
   1:  PR[91,2] = PR[90,2] + 8.300;
   1:L PR[91] R[100]mm/sec CNT100;
   1:  PR[91,1] = PR[90,1] + -38.933;
   1:  PR[91,2] = PR[90,2] + 4.458;
   1:L PR[91] R[100]mm/sec CNT100;
   1:  PR[91,1] = PR[90,1] + -38.984;
   1:  PR[91,2] = PR[90,2] + 4.258;
   1:L PR[91] R[100]mm/sec CNT100;
   1:  PR[91,1] = PR[90,1] + -39.549;
   1:  PR[91,2] = PR[90,2] + -0.193;
   1:L PR[91] R[100]mm/sec CNT100;
   1:  PR[91,1] = PR[90,1] + -39.555;
   1:  PR[91,2] = PR[90,2] + -0.277;
   1:L PR[91] R[100]mm/sec CNT100;
   1:  PR[91,1] = PR[90,1] + -38.998;
   1:  PR[91,2] = PR[90,2] + -4.626;
   1:L PR[91] R[100]mm/sec CNT100;
   1:  PR[91,1] = PR[90,1] + -38.976;
   1:  PR[91,2] = PR[90,2] + -4.916;
   1:L PR[91] R[100]mm/sec CNT100;
   1:  PR[91,1] = PR[90,1] + -38.933;
   1:  PR[91,2] = PR[90,2] + -5.082;
   1:L PR[91] R[100]mm/sec CNT100;
   1:  PR[91,1] = PR[90,1] + -37.391;
   1:  PR[91,2] = PR[90,2] + -8.924;
   1:L PR[91] R[100]mm/sec CNT100;
   1:  PR[91,1] = PR[90,1] + -37.221;
   1:  PR[91,2] = PR[90,2] + -9.304;
   1:L PR[91] R[100]mm/sec CNT100;
   1:  PR[91,1] = PR[90,1] + -35.013;
   1:  PR[91,2] = PR[90,2] + -12.368;
   1:L PR[91] R[100]mm/sec CNT100;
   1:  PR[91,1] = PR[90,1] + -34.612;
   1:  PR[91,2] = PR[90,2] + -12.985;
   1:L PR[91] R[100]mm/sec CNT100;
   1:  PR[91,1] = PR[90,1] + -34.108;
   1:  PR[91,2] = PR[90,2] + -13.528;
   1:L PR[91] R[100]mm/sec CNT100;
   1:  PR[91,1] = PR[90,1] + -31.597;
   1:  PR[91,2] = PR[90,2] + -15.658;
   1:L PR[91] R[100]mm/sec CNT100;
   1:  PR[91,1] = PR[90,1] + -30.685;
   1:  PR[91,2] = PR[90,2] + -16.371;
   1:L PR[91] R[100]mm/sec CNT100;
   1:  PR[91,1] = PR[90,1] + -29.329;
   1:  PR[91,2] = PR[90,2] + -17.123;
   1:L PR[91] R[100]mm/sec CNT100;
   1:  PR[91,1] = PR[90,1] + -27.094;
   1:  PR[91,2] = PR[90,2] + -18.253;
   1:L PR[91] R[100]mm/sec CNT100;
   1:  PR[91,1] = PR[90,1] + -25.249;
   1:  PR[91,2] = PR[90,2] + -18.923;
   1:L PR[91] R[100]mm/sec CNT100;
   1:  PR[91,1] = PR[90,1] + -23.709;
   1:  PR[91,2] = PR[90,2] + -19.293;
   1:L PR[91] R[100]mm/sec CNT100;
   1:  PR[91,1] = PR[90,1] + -21.400;
   1:  PR[91,2] = PR[90,2] + -19.753;
   1:L PR[91] R[100]mm/sec CNT100;
   1:  PR[91,1] = PR[90,1] + -18.017;
   1:  PR[91,2] = PR[90,2] + -19.893;
   1:L PR[91] R[100]mm/sec CNT100;
   1:  PR[91,1] = PR[90,1] + -14.772;
   1:  PR[91,2] = PR[90,2] + -19.561;
   1:L PR[91] R[100]mm/sec CNT100;
   1:  PR[91,1] = PR[90,1] + -14.588;
   1:  PR[91,2] = PR[90,2] + -19.535;
   1:L PR[91] R[100]mm/sec CNT100;
   1:  PR[91,1] = PR[90,1] + -11.527;
   1:  PR[91,2] = PR[90,2] + -18.744;
   1:L PR[91] R[100]mm/sec CNT100;
   1:  PR[91,1] = PR[90,1] + -8.132;
   1:  PR[91,2] = PR[90,2] + -17.265;
   1:L PR[91] R[100]mm/sec CNT100;
   1:  PR[91,1] = PR[90,1] + -5.792;
   1:  PR[91,2] = PR[90,2] + -15.768;
   1:L PR[91] R[100]mm/sec CNT100;
   1:  PR[91,1] = PR[90,1] + -5.572;
   1:  PR[91,2] = PR[90,2] + -15.609;
   1:L PR[91] R[100]mm/sec CNT100;
   1:  PR[91,1] = PR[90,1] + -4.695;
   1:  PR[91,2] = PR[90,2] + -14.841;
   1:L PR[91] R[100]mm/sec CNT100;
   1:  PR[91,1] = PR[90,1] + -3.391;
   1:  PR[91,2] = PR[90,2] + -13.666;
   1:L PR[91] R[100]mm/sec CNT100;
   1:  PR[91,1] = PR[90,1] + -2.151;
   1:  PR[91,2] = PR[90,2] + -12.212;
   1:L PR[91] R[100]mm/sec CNT100;
   1:  PR[91,1] = PR[90,1] + -0.583;
   1:  PR[91,2] = PR[90,2] + -11.079;
   1:L PR[91] R[100]mm/sec CNT100;
   1:  PR[91,1] = PR[90,1] + 0.069;
   1:  PR[91,2] = PR[90,2] + -11.311;
   1:L PR[91] R[100]mm/sec CNT100;
   1:  PR[91,1] = PR[90,1] + 1.073;
   1:L PR[91] R[100]mm/sec CNT100;
   1:  PR[91,1] = PR[90,1] + 2.317;
   1:  PR[91,2] = PR[90,2] + -12.214;
   1:L PR[91] R[100]mm/sec CNT100;
   1:  PR[91,1] = PR[90,1] + 3.564;
   1:  PR[91,2] = PR[90,2] + -13.680;
   1:L PR[91] R[100]mm/sec CNT100;
   1:  PR[91,1] = PR[90,1] + 4.868;
   1:  PR[91,2] = PR[90,2] + -14.855;
   1:L PR[91] R[100]mm/sec CNT100;
   1:  PR[91,1] = PR[90,1] + 5.716;
   1:  PR[91,2] = PR[90,2] + -15.599;
   1:L PR[91] R[100]mm/sec CNT100;
   1:  PR[91,1] = PR[90,1] + 7.989;
   1:  PR[91,2] = PR[90,2] + -17.055;
   1:L PR[91] R[100]mm/sec CNT100;
   1:  PR[91,1] = PR[90,1] + 8.308;
   1:  PR[91,2] = PR[90,2] + -17.275;
   1:L PR[91] R[100]mm/sec CNT100;
   1:  PR[91,1] = PR[90,1] + 11.676;
   1:  PR[91,2] = PR[90,2] + -18.739;
   1:L PR[91] R[100]mm/sec CNT100;
   1:  PR[91,1] = PR[90,1] + 14.718;
   1:  PR[91,2] = PR[90,2] + -19.527;
   1:L PR[91] R[100]mm/sec CNT100;
   1:  PR[91,1] = PR[90,1] + 18.167;
   1:  PR[91,2] = PR[90,2] + -19.893;
   1:L PR[91] R[100]mm/sec CNT100;
   1:  PR[91,1] = PR[90,1] + 21.512;
   1:  PR[91,2] = PR[90,2] + -19.757;
   1:L PR[91] R[100]mm/sec CNT100;
   1:  PR[91,1] = PR[90,1] + 22.570;
   1:  PR[91,2] = PR[90,2] + -19.507;
   1:L PR[91] R[100]mm/sec CNT100;
   1:  PR[91,1] = PR[90,1] + 25.408;
   1:  PR[91,2] = PR[90,2] + -18.919;
   1:L PR[91] R[100]mm/sec CNT100;
   1:  PR[91,1] = PR[90,1] + 27.241;
   1:  PR[91,2] = PR[90,2] + -18.257;
   1:L PR[91] R[100]mm/sec CNT100;
   1:  PR[91,1] = PR[90,1] + 29.476;
   1:  PR[91,2] = PR[90,2] + -17.129;
   1:L PR[91] R[100]mm/sec CNT100;
   1:  PR[91,1] = PR[90,1] + 30.806;
   1:  PR[91,2] = PR[90,2] + -16.395;
   1:L PR[91] R[100]mm/sec CNT100;
   1:  PR[91,1] = PR[90,1] + 33.387;
   1:  PR[91,2] = PR[90,2] + -14.216;
   1:L PR[91] R[100]mm/sec CNT100;
   1:  PR[91,1] = PR[90,1] + 34.268;
   1:  PR[91,2] = PR[90,2] + -13.521;
   1:L PR[91] R[100]mm/sec CNT100;
   1:  PR[91,1] = PR[90,1] + 34.781;
   1:  PR[91,2] = PR[90,2] + -12.969;
   1:L PR[91] R[100]mm/sec CNT100;
   1:  PR[91,1] = PR[90,1] + 37.072;
   1:  PR[91,2] = PR[90,2] + -9.770;
   1:L PR[91] R[100]mm/sec CNT100;
   1:  PR[91,1] = PR[90,1] + 37.365;
   1:  PR[91,2] = PR[90,2] + -9.327;
   1:L PR[91] R[100]mm/sec CNT100;
   1:  PR[91,1] = PR[90,1] + 37.546;
   1:  PR[91,2] = PR[90,2] + -8.925;
   1:L PR[91] R[100]mm/sec CNT100;
   1:  PR[91,1] = PR[90,1] + 39.088;
   1:  PR[91,2] = PR[90,2] + -5.103;
   1:L PR[91] R[100]mm/sec CNT100;
   1:  PR[91,1] = PR[90,1] + 39.140;
   1:  PR[91,2] = PR[90,2] + -4.908;
   1:L PR[91] R[100]mm/sec CNT100;
   1:  PR[91,1] = PR[90,1] + 39.704;
   1:  PR[91,2] = PR[90,2] + -0.438;
   1:L PR[91] R[100]mm/sec CNT100;
   1:  PR[91,1] = PR[90,1] + 39.712;
   1:  PR[91,2] = PR[90,2] + -0.345;
   1:L PR[91] R[100]mm/sec CNT100;
   1:  PR[91,1] = PR[90,1] + 39.155;
   1:  PR[91,2] = PR[90,2] + 4.019;
   1:L PR[91] R[100]mm/sec CNT100;
   1:  PR[91,1] = PR[90,1] + 39.131;
   1:  PR[91,2] = PR[90,2] + 4.317;
   1:L PR[91] R[100]mm/sec CNT100;
   1:  PR[91,1] = PR[90,1] + 39.088;
   1:  PR[91,2] = PR[90,2] + 4.480;
   1:L PR[91] R[100]mm/sec CNT100;
   1:  PR[91,1] = PR[90,1] + 37.545;
   1:  PR[91,2] = PR[90,2] + 8.303;
   1:L PR[91] R[100]mm/sec CNT100;
   1:  PR[91,1] = PR[90,1] + 37.376;
   1:  PR[91,2] = PR[90,2] + 8.678;
   1:L PR[91] R[100]mm/sec CNT100;
   1:  PR[91,1] = PR[90,1] + 35.166;
   1:  PR[91,2] = PR[90,2] + 11.747;
   1:L PR[91] R[100]mm/sec CNT100;
   1:  PR[91,1] = PR[90,1] + 34.758;
   1:  PR[91,2] = PR[90,2] + 12.370;
   1:L PR[91] R[100]mm/sec CNT100;
   1:  PR[91,1] = PR[90,1] + 34.247;
   1:  PR[91,2] = PR[90,2] + 12.919;
   1:L PR[91] R[100]mm/sec CNT100;
   1:  PR[91,1] = PR[90,1] + 31.735;
   1:  PR[91,2] = PR[90,2] + 15.054;
   1:L PR[91] R[100]mm/sec CNT100;
   1:  PR[91,1] = PR[90,1] + 30.828;
   1:  PR[91,2] = PR[90,2] + 15.759;
   1:L PR[91] R[100]mm/sec CNT100;
   1:  PR[91,1] = PR[90,1] + 29.473;
   1:  PR[91,2] = PR[90,2] + 16.507;
   1:L PR[91] R[100]mm/sec CNT100;
   1:  PR[91,1] = PR[90,1] + 27.238;
   1:  PR[91,2] = PR[90,2] + 17.634;
   1:L PR[91] R[100]mm/sec CNT100;
   1:  PR[91,1] = PR[90,1] + 25.384;
   1:  PR[91,2] = PR[90,2] + 18.304;
   1:L PR[91] R[100]mm/sec CNT100;
   1:  PR[91,1] = PR[90,1] + 23.847;
   1:  PR[91,2] = PR[90,2] + 18.673;
   1:L PR[91] R[100]mm/sec CNT100;
   1:  PR[91,1] = PR[90,1] + 21.536;
   1:  PR[91,2] = PR[90,2] + 19.132;
   1:L PR[91] R[100]mm/sec CNT100;
   1:  PR[91,1] = PR[90,1] + 18.167;
   1:  PR[91,2] = PR[90,2] + 19.269;
   1:L PR[91] R[100]mm/sec CNT100;
   1:  PR[91,1] = PR[90,1] + 14.720;
   1:  PR[91,2] = PR[90,2] + 18.904;
   1:L PR[91] R[100]mm/sec CNT100;
   1:  PR[91,1] = PR[90,1] + 11.682;
   1:  PR[91,2] = PR[90,2] + 18.117;
   1:L PR[91] R[100]mm/sec CNT100;
   1:  PR[91,1] = PR[90,1] + 9.005;
   1:  PR[91,2] = PR[90,2] + 16.945;
   1:L PR[91] R[100]mm/sec CNT100;
   1:  PR[91,1] = PR[90,1] + 8.300;
   1:  PR[91,2] = PR[90,2] + 16.651;
   1:L PR[91] R[100]mm/sec CNT100;
   1:  PR[91,1] = PR[90,1] + 5.972;
   1:  PR[91,2] = PR[90,2] + 15.164;
   1:L PR[91] R[100]mm/sec CNT100;
   1:  PR[91,1] = PR[90,1] + 5.833;
   1:  PR[91,2] = PR[90,2] + 15.068;
   1:L PR[91] R[100]mm/sec CNT100;
   1:  PR[91,1] = PR[90,1] + 5.556;
   1:  PR[91,2] = PR[90,2] + 14.849;
   1:L PR[91] R[100]mm/sec CNT100;
   1:  PR[91,1] = PR[90,1] + 3.621;
   1:  PR[91,2] = PR[90,2] + 13.113;
   1:L PR[91] R[100]mm/sec CNT100;
   1:  PR[91,1] = PR[90,1] + 3.087;
   1:  PR[91,2] = PR[90,2] + 12.552;
   1:L PR[91] R[100]mm/sec CNT100;
   1:  PR[91,1] = PR[90,1] + 2.482;
   1:  PR[91,2] = PR[90,2] + 11.783;
   1:L PR[91] R[100]mm/sec CNT100;
   1:  PR[91,1] = PR[90,1] + 2.387;
   1:  PR[91,2] = PR[90,2] + 11.701;
   1:L PR[91] R[100]mm/sec CNT100;
   1:  PR[91,1] = PR[90,1] + 2.261;
   1:  PR[91,2] = PR[90,2] + 11.536;
   1:L PR[91] R[100]mm/sec CNT100;
   1:  PR[91,1] = PR[90,1] + 1.369;
   1:  PR[91,2] = PR[90,2] + 10.904;
   1:L PR[91] R[100]mm/sec CNT100;
   1:  PR[91,1] = PR[90,1] + 0.860;
   1:  PR[91,2] = PR[90,2] + 10.625;
   1:L PR[91] R[100]mm/sec CNT100;
   1:  PR[91,1] = PR[90,1] + -0.659;
   1:L PR[91] R[100]mm/sec CNT100;
   1:  PR[91] = PR[90];
   1:  PR[91,1] = PR[90,1] + -1.423;
   1:  PR[91,2] = PR[90,2] + 11.291;
   1:  PR[91,3] = PR[90,3] + 26.535;
   1:L PR[91] R[100]mm/sec CNT100;
   1:  PR[91,1] = PR[90,1] + -1.660;
   1:  PR[91,2] = PR[90,2] + 11.599;
   1:L PR[91] R[100]mm/sec CNT100;
   1:  PR[91,1] = PR[90,1] + -1.793;
   1:  PR[91,2] = PR[90,2] + 11.725;
   1:L PR[91] R[100]mm/sec CNT100;
   1:  PR[91,1] = PR[90,1] + -2.139;
   1:  PR[91,2] = PR[90,2] + 11.974;
   1:L PR[91] R[100]mm/sec CNT100;
   1:  PR[91,1] = PR[90,1] + -2.612;
   1:  PR[91,2] = PR[90,2] + 12.543;
   1:L PR[91] R[100]mm/sec CNT100;
   1:  PR[91,1] = PR[90,1] + -3.255;
   1:  PR[91,2] = PR[90,2] + 13.216;
   1:L PR[91] R[100]mm/sec CNT100;
   1:  PR[91,1] = PR[90,1] + -5.096;
   1:  PR[91,2] = PR[90,2] + 14.865;
   1:L PR[91] R[100]mm/sec CNT100;
   1:  PR[91,1] = PR[90,1] + -5.421;
   1:  PR[91,2] = PR[90,2] + 15.121;
   1:L PR[91] R[100]mm/sec CNT100;
   1:  PR[91,1] = PR[90,1] + -7.872;
   1:  PR[91,2] = PR[90,2] + 16.700;
   1:L PR[91] R[100]mm/sec CNT100;
   1:  PR[91,1] = PR[90,1] + -10.624;
   1:  PR[91,2] = PR[90,2] + 17.903;
   1:L PR[91] R[100]mm/sec CNT100;
   1:  PR[91,1] = PR[90,1] + -11.327;
   1:  PR[91,2] = PR[90,2] + 18.197;
   1:L PR[91] R[100]mm/sec CNT100;
   1:  PR[91,1] = PR[90,1] + -14.242;
   1:  PR[91,2] = PR[90,2] + 18.951;
   1:L PR[91] R[100]mm/sec CNT100;
   1:  PR[91,1] = PR[90,1] + -17.828;
   1:  PR[91,2] = PR[90,2] + 19.331;
   1:L PR[91] R[100]mm/sec CNT100;
   1:  PR[91,1] = PR[90,1] + -21.174;
   1:  PR[91,2] = PR[90,2] + 19.169;
   1:L PR[91] R[100]mm/sec CNT100;
   1:  PR[91,1] = PR[90,1] + -21.521;
   1:  PR[91,2] = PR[90,2] + 19.087;
   1:L PR[91] R[100]mm/sec CNT100;
   1:  PR[91,1] = PR[90,1] + -24.881;
   1:  PR[91,2] = PR[90,2] + 18.390;
   1:L PR[91] R[100]mm/sec CNT100;
   1:  PR[91,1] = PR[90,1] + -27.068;
   1:  PR[91,2] = PR[90,2] + 17.595;
   1:L PR[91] R[100]mm/sec CNT100;
   1:  PR[91,1] = PR[90,1] + -28.779;
   1:  PR[91,2] = PR[90,2] + 16.730;
   1:L PR[91] R[100]mm/sec CNT100;
   1:  PR[91,1] = PR[90,1] + -30.477;
   1:  PR[91,2] = PR[90,2] + 15.788;
   1:L PR[91] R[100]mm/sec CNT100;
   1:  PR[91,1] = PR[90,1] + -32.592;
   1:  PR[91,2] = PR[90,2] + 14.005;
   1:L PR[91] R[100]mm/sec CNT100;
   1:  PR[91,1] = PR[90,1] + -33.817;
   1:  PR[91,2] = PR[90,2] + 13.036;
   1:L PR[91] R[100]mm/sec CNT100;
   1:  PR[91,1] = PR[90,1] + -34.559;
   1:  PR[91,2] = PR[90,2] + 12.238;
   1:L PR[91] R[100]mm/sec CNT100;
   1:  PR[91,1] = PR[90,1] + -36.546;
   1:  PR[91,2] = PR[90,2] + 9.463;
   1:L PR[91] R[100]mm/sec CNT100;
   1:  PR[91,1] = PR[90,1] + -37.031;
   1:  PR[91,2] = PR[90,2] + 8.726;
   1:L PR[91] R[100]mm/sec CNT100;
   1:  PR[91,1] = PR[90,1] + -37.345;
   1:  PR[91,2] = PR[90,2] + 8.022;
   1:L PR[91] R[100]mm/sec CNT100;
   1:  PR[91,1] = PR[90,1] + -38.715;
   1:  PR[91,2] = PR[90,2] + 4.608;
   1:L PR[91] R[100]mm/sec CNT100;
   1:  PR[91,1] = PR[90,1] + -38.845;
   1:  PR[91,2] = PR[90,2] + 4.104;
   1:L PR[91] R[100]mm/sec CNT100;
   1:  PR[91,1] = PR[90,1] + -39.349;
   1:  PR[91,2] = PR[90,2] + 0.130;
   1:L PR[91] R[100]mm/sec CNT100;
   1:  PR[91,1] = PR[90,1] + -39.381;
   1:  PR[91,2] = PR[90,2] + -0.277;
   1:L PR[91] R[100]mm/sec CNT100;
   1:  PR[91,1] = PR[90,1] + -38.883;
   1:  PR[91,2] = PR[90,2] + -4.167;
   1:L PR[91] R[100]mm/sec CNT100;
   1:  PR[91,1] = PR[90,1] + -38.837;
   1:  PR[91,2] = PR[90,2] + -4.762;
   1:L PR[91] R[100]mm/sec CNT100;
   1:  PR[91,1] = PR[90,1] + -38.715;
   1:  PR[91,2] = PR[90,2] + -5.232;
   1:L PR[91] R[100]mm/sec CNT100;
   1:  PR[91,1] = PR[90,1] + -37.344;
   1:  PR[91,2] = PR[90,2] + -8.646;
   1:L PR[91] R[100]mm/sec CNT100;
   1:  PR[91,1] = PR[90,1] + -37.044;
   1:  PR[91,2] = PR[90,2] + -9.321;
   1:L PR[91] R[100]mm/sec CNT100;
   1:  PR[91,1] = PR[90,1] + -35.099;
   1:  PR[91,2] = PR[90,2] + -12.020;
   1:L PR[91] R[100]mm/sec CNT100;
   1:  PR[91,1] = PR[90,1] + -34.536;
   1:  PR[91,2] = PR[90,2] + -12.886;
   1:L PR[91] R[100]mm/sec CNT100;
   1:  PR[91,1] = PR[90,1] + -33.800;
   1:  PR[91,2] = PR[90,2] + -13.678;
   1:L PR[91] R[100]mm/sec CNT100;
   1:  PR[91,1] = PR[90,1] + -31.666;
   1:  PR[91,2] = PR[90,2] + -15.488;
   1:L PR[91] R[100]mm/sec CNT100;
   1:  PR[91,1] = PR[90,1] + -30.501;
   1:  PR[91,2] = PR[90,2] + -16.399;
   1:L PR[91] R[100]mm/sec CNT100;
   1:  PR[91,1] = PR[90,1] + -28.778;
   1:  PR[91,2] = PR[90,2] + -17.354;
   1:L PR[91] R[100]mm/sec CNT100;
   1:  PR[91,1] = PR[90,1] + -27.068;
   1:  PR[91,2] = PR[90,2] + -18.219;
   1:L PR[91] R[100]mm/sec CNT100;
   1:  PR[91,1] = PR[90,1] + -24.860;
   1:  PR[91,2] = PR[90,2] + -19.021;
   1:L PR[91] R[100]mm/sec CNT100;
   1:  PR[91,1] = PR[90,1] + -23.856;
   1:  PR[91,2] = PR[90,2] + -19.262;
   1:L PR[91] R[100]mm/sec CNT100;
   1:  PR[91,1] = PR[90,1] + -21.199;
   1:  PR[91,2] = PR[90,2] + -19.791;
   1:L PR[91] R[100]mm/sec CNT100;
   1:  PR[91,1] = PR[90,1] + -17.823;
   1:  PR[91,2] = PR[90,2] + -19.955;
   1:L PR[91] R[100]mm/sec CNT100;
   1:  PR[91,1] = PR[90,1] + -14.672;
   1:  PR[91,2] = PR[90,2] + -19.637;
   1:L PR[91] R[100]mm/sec CNT100;
   1:  PR[91,1] = PR[90,1] + -14.261;
   1:  PR[91,2] = PR[90,2] + -19.580;
   1:L PR[91] R[100]mm/sec CNT100;
   1:  PR[91,1] = PR[90,1] + -11.329;
   1:  PR[91,2] = PR[90,2] + -18.822;
   1:L PR[91] R[100]mm/sec CNT100;
   1:  PR[91,1] = PR[90,1] + -7.839;
   1:  PR[91,2] = PR[90,2] + -17.303;
   1:L PR[91] R[100]mm/sec CNT100;
   1:  PR[91,1] = PR[90,1] + -5.607;
   1:  PR[91,2] = PR[90,2] + -15.876;
   1:L PR[91] R[100]mm/sec CNT100;
   1:  PR[91,1] = PR[90,1] + -5.328;
   1:  PR[91,2] = PR[90,2] + -15.675;
   1:L PR[91] R[100]mm/sec CNT100;
   1:  PR[91,1] = PR[90,1] + -4.271;
   1:  PR[91,2] = PR[90,2] + -14.749;
   1:L PR[91] R[100]mm/sec CNT100;
   1:  PR[91,1] = PR[90,1] + -3.185;
   1:  PR[91,2] = PR[90,2] + -13.771;
   1:L PR[91] R[100]mm/sec CNT100;
   1:  PR[91,1] = PR[90,1] + -2.156;
   1:  PR[91,2] = PR[90,2] + -12.565;
   1:L PR[91] R[100]mm/sec CNT100;
   1:  PR[91,1] = PR[90,1] + -1.829;
   1:  PR[91,2] = PR[90,2] + -12.302;
   1:L PR[91] R[100]mm/sec CNT100;
   1:  PR[91,1] = PR[90,1] + -0.550;
   1:  PR[91,2] = PR[90,2] + -11.397;
   1:L PR[91] R[100]mm/sec CNT100;
   1:  PR[91,1] = PR[90,1] + 0.193;
   1:  PR[91,2] = PR[90,2] + -11.661;
   1:L PR[91] R[100]mm/sec CNT100;
   1:  PR[91,1] = PR[90,1] + 1.144;
   1:L PR[91] R[100]mm/sec CNT100;
   1:  PR[91,1] = PR[90,1] + 1.657;
   1:  PR[91,2] = PR[90,2] + -12.081;
   1:L PR[91] R[100]mm/sec CNT100;
   1:  PR[91,1] = PR[90,1] + 2.294;
   1:  PR[91,2] = PR[90,2] + -12.534;
   1:L PR[91] R[100]mm/sec CNT100;
   1:  PR[91,1] = PR[90,1] + 3.356;
   1:  PR[91,2] = PR[90,2] + -13.783;
   1:L PR[91] R[100]mm/sec CNT100;
   1:  PR[91,1] = PR[90,1] + 4.441;
   1:  PR[91,2] = PR[90,2] + -14.761;
   1:L PR[91] R[100]mm/sec CNT100;
   1:  PR[91,1] = PR[90,1] + 5.471;
   1:  PR[91,2] = PR[90,2] + -15.664;
   1:L PR[91] R[100]mm/sec CNT100;
   1:  PR[91,1] = PR[90,1] + 7.593;
   1:  PR[91,2] = PR[90,2] + -17.023;
   1:L PR[91] R[100]mm/sec CNT100;
   1:  PR[91,1] = PR[90,1] + 8.015;
   1:  PR[91,2] = PR[90,2] + -17.314;
   1:L PR[91] R[100]mm/sec CNT100;
   1:  PR[91,1] = PR[90,1] + 11.478;
   1:  PR[91,2] = PR[90,2] + -18.817;
   1:L PR[91] R[100]mm/sec CNT100;
   1:  PR[91,1] = PR[90,1] + 14.391;
   1:  PR[91,2] = PR[90,2] + -19.572;
   1:L PR[91] R[100]mm/sec CNT100;
   1:  PR[91,1] = PR[90,1] + 17.974;
   1:  PR[91,2] = PR[90,2] + -19.955;
   1:L PR[91] R[100]mm/sec CNT100;
   1:  PR[91,1] = PR[90,1] + 21.307;
   1:  PR[91,2] = PR[90,2] + -19.796;
   1:L PR[91] R[100]mm/sec CNT100;
   1:  PR[91,1] = PR[90,1] + 21.648;
   1:  PR[91,2] = PR[90,2] + -19.716;
   1:L PR[91] R[100]mm/sec CNT100;
   1:  PR[91,1] = PR[90,1] + 25.016;
   1:  PR[91,2] = PR[90,2] + -19.018;
   1:L PR[91] R[100]mm/sec CNT100;
   1:  PR[91,1] = PR[90,1] + 27.213;
   1:  PR[91,2] = PR[90,2] + -18.224;
   1:L PR[91] R[100]mm/sec CNT100;
   1:  PR[91,1] = PR[90,1] + 28.922;
   1:  PR[91,2] = PR[90,2] + -17.361;
   1:L PR[91] R[100]mm/sec CNT100;
   1:  PR[91,1] = PR[90,1] + 30.618;
   1:  PR[91,2] = PR[90,2] + -16.426;
   1:L PR[91] R[100]mm/sec CNT100;
   1:  PR[91,1] = PR[90,1] + 32.732;
   1:  PR[91,2] = PR[90,2] + -14.641;
   1:L PR[91] R[100]mm/sec CNT100;
   1:  PR[91,1] = PR[90,1] + 33.954;
   1:  PR[91,2] = PR[90,2] + -13.677;
   1:L PR[91] R[100]mm/sec CNT100;
   1:  PR[91,1] = PR[90,1] + 34.702;
   1:  PR[91,2] = PR[90,2] + -12.874;
   1:L PR[91] R[100]mm/sec CNT100;
   1:  PR[91,1] = PR[90,1] + 36.691;
   1:  PR[91,2] = PR[90,2] + -10.095;
   1:L PR[91] R[100]mm/sec CNT100;
   1:  PR[91,1] = PR[90,1] + 37.186;
   1:  PR[91,2] = PR[90,2] + -9.346;
   1:L PR[91] R[100]mm/sec CNT100;
   1:  PR[91,1] = PR[90,1] + 37.499;
   1:  PR[91,2] = PR[90,2] + -8.654;
   1:L PR[91] R[100]mm/sec CNT100;
   1:  PR[91,1] = PR[90,1] + 38.869;
   1:  PR[91,2] = PR[90,2] + -5.258;
   1:L PR[91] R[100]mm/sec CNT100;
   1:  PR[91,1] = PR[90,1] + 38.999;
   1:  PR[91,2] = PR[90,2] + -4.762;
   1:L PR[91] R[100]mm/sec CNT100;
   1:  PR[91,1] = PR[90,1] + 39.503;
   1:  PR[91,2] = PR[90,2] + -0.771;
   1:L PR[91] R[100]mm/sec CNT100;
   1:  PR[91,1] = PR[90,1] + 39.538;
   1:  PR[91,2] = PR[90,2] + -0.345;
   1:L PR[91] R[100]mm/sec CNT100;
   1:  PR[91,1] = PR[90,1] + 39.040;
   1:  PR[91,2] = PR[90,2] + 3.557;
   1:L PR[91] R[100]mm/sec CNT100;
   1:  PR[91,1] = PR[90,1] + 38.991;
   1:  PR[91,2] = PR[90,2] + 4.171;
   1:L PR[91] R[100]mm/sec CNT100;
   1:  PR[91,1] = PR[90,1] + 38.869;
   1:  PR[91,2] = PR[90,2] + 4.635;
   1:L PR[91] R[100]mm/sec CNT100;
   1:  PR[91,1] = PR[90,1] + 37.498;
   1:  PR[91,2] = PR[90,2] + 8.032;
   1:L PR[91] R[100]mm/sec CNT100;
   1:  PR[91,1] = PR[90,1] + 37.197;
   1:  PR[91,2] = PR[90,2] + 8.698;
   1:L PR[91] R[100]mm/sec CNT100;
   1:  PR[91,1] = PR[90,1] + 35.251;
   1:  PR[91,2] = PR[90,2] + 11.401;
   1:L PR[91] R[100]mm/sec CNT100;
   1:  PR[91,1] = PR[90,1] + 34.679;
   1:  PR[91,2] = PR[90,2] + 12.274;
   1:L PR[91] R[100]mm/sec CNT100;
   1:  PR[91,1] = PR[90,1] + 33.934;
   1:  PR[91,2] = PR[90,2] + 13.074;
   1:L PR[91] R[100]mm/sec CNT100;
   1:  PR[91,1] = PR[90,1] + 31.800;
   1:  PR[91,2] = PR[90,2] + 14.887;
   1:L PR[91] R[100]mm/sec CNT100;
   1:  PR[91,1] = PR[90,1] + 30.641;
   1:  PR[91,2] = PR[90,2] + 15.790;
   1:L PR[91] R[100]mm/sec CNT100;
   1:  PR[91,1] = PR[90,1] + 28.920;
   1:  PR[91,2] = PR[90,2] + 16.738;
   1:L PR[91] R[100]mm/sec CNT100;
   1:  PR[91,1] = PR[90,1] + 27.211;
   1:  PR[91,2] = PR[90,2] + 17.600;
   1:L PR[91] R[100]mm/sec CNT100;
   1:  PR[91,1] = PR[90,1] + 24.993;
   1:  PR[91,2] = PR[90,2] + 18.402;
   1:L PR[91] R[100]mm/sec CNT100;
   1:  PR[91,1] = PR[90,1] + 23.992;
   1:  PR[91,2] = PR[90,2] + 18.642;
   1:L PR[91] R[100]mm/sec CNT100;
   1:  PR[91,1] = PR[90,1] + 21.332;
   1:  PR[91,2] = PR[90,2] + 19.171;
   1:L PR[91] R[100]mm/sec CNT100;
   1:  PR[91,1] = PR[90,1] + 17.971;
   1:  PR[91,2] = PR[90,2] + 19.331;
   1:L PR[91] R[100]mm/sec CNT100;
   1:  PR[91,1] = PR[90,1] + 14.829;
   1:  PR[91,2] = PR[90,2] + 19.012;
   1:L PR[91] R[100]mm/sec CNT100;
   1:  PR[91,1] = PR[90,1] + 14.418;
   1:  PR[91,2] = PR[90,2] + 18.955;
   1:L PR[91] R[100]mm/sec CNT100;
   1:  PR[91,1] = PR[90,1] + 11.487;
   1:  PR[91,2] = PR[90,2] + 18.196;
   1:L PR[91] R[100]mm/sec CNT100;
   1:  PR[91,1] = PR[90,1] + 8.920;
   1:  PR[91,2] = PR[90,2] + 17.072;
   1:L PR[91] R[100]mm/sec CNT100;
   1:  PR[91,1] = PR[90,1] + 8.012;
   1:  PR[91,2] = PR[90,2] + 16.693;
   1:L PR[91] R[100]mm/sec CNT100;
   1:  PR[91,1] = PR[90,1] + 5.789;
   1:  PR[91,2] = PR[90,2] + 15.274;
   1:L PR[91] R[100]mm/sec CNT100;
   1:  PR[91,1] = PR[90,1] + 5.612;
   1:  PR[91,2] = PR[90,2] + 15.152;
   1:L PR[91] R[100]mm/sec CNT100;
   1:  PR[91,1] = PR[90,1] + 5.268;
   1:  PR[91,2] = PR[90,2] + 14.879;
   1:L PR[91] R[100]mm/sec CNT100;
   1:  PR[91,1] = PR[90,1] + 3.427;
   1:  PR[91,2] = PR[90,2] + 13.229;
   1:L PR[91] R[100]mm/sec CNT100;
   1:  PR[91,1] = PR[90,1] + 2.786;
   1:  PR[91,2] = PR[90,2] + 12.556;
   1:L PR[91] R[100]mm/sec CNT100;
   1:  PR[91,1] = PR[90,1] + 2.184;
   1:  PR[91,2] = PR[90,2] + 11.814;
   1:L PR[91] R[100]mm/sec CNT100;
   1:  PR[91,1] = PR[90,1] + 1.393;
   1:  PR[91,2] = PR[90,2] + 11.254;
   1:L PR[91] R[100]mm/sec CNT100;
   1:  PR[91,1] = PR[90,1] + 0.820;
   1:  PR[91,2] = PR[90,2] + 10.940;
   1:L PR[91] R[100]mm/sec CNT100;
   1:  PR[91,1] = PR[90,1] + -0.635;
   1:L PR[91] R[100]mm/sec CNT100;
   1:  PR[91] = PR[90];
   1:  PR[91,1] = PR[90,1] + -1.462;
   1:  PR[91,2] = PR[90,2] + 11.634;
   1:  PR[91,3] = PR[90,3] + 27.145;
   1:L PR[91] R[100]mm/sec CNT100;
   1:  PR[91,1] = PR[90,1] + -1.730;
   1:  PR[91,2] = PR[90,2] + 11.982;
   1:L PR[91] R[100]mm/sec CNT100;
   1:  PR[91,1] = PR[90,1] + -1.967;
   1:  PR[91,2] = PR[90,2] + 12.206;
   1:L PR[91] R[100]mm/sec CNT100;
   1:  PR[91,1] = PR[90,1] + -2.120;
   1:  PR[91,2] = PR[90,2] + 12.316;
   1:L PR[91] R[100]mm/sec CNT100;
   1:  PR[91,1] = PR[90,1] + -2.321;
   1:  PR[91,2] = PR[90,2] + 12.557;
   1:L PR[91] R[100]mm/sec CNT100;
   1:  PR[91,1] = PR[90,1] + -3.063;
   1:  PR[91,2] = PR[90,2] + 13.334;
   1:L PR[91] R[100]mm/sec CNT100;
   1:  PR[91,1] = PR[90,1] + -4.810;
   1:  PR[91,2] = PR[90,2] + 14.896;
   1:L PR[91] R[100]mm/sec CNT100;
   1:  PR[91,1] = PR[90,1] + -5.202;
   1:  PR[91,2] = PR[90,2] + 15.206;
   1:L PR[91] R[100]mm/sec CNT100;
   1:  PR[91,1] = PR[90,1] + -7.585;
   1:  PR[91,2] = PR[90,2] + 16.743;
   1:L PR[91] R[100]mm/sec CNT100;
   1:  PR[91,1] = PR[90,1] + -10.209;
   1:  PR[91,2] = PR[90,2] + 17.890;
   1:L PR[91] R[100]mm/sec CNT100;
   1:  PR[91,1] = PR[90,1] + -11.131;
   1:  PR[91,2] = PR[90,2] + 18.276;
   1:L PR[91] R[100]mm/sec CNT100;
   1:  PR[91,1] = PR[90,1] + -13.916;
   1:  PR[91,2] = PR[90,2] + 18.996;
   1:L PR[91] R[100]mm/sec CNT100;
   1:  PR[91,1] = PR[90,1] + -17.278;
   1:  PR[91,2] = PR[90,2] + 19.346;
   1:L PR[91] R[100]mm/sec CNT100;
   1:  PR[91,1] = PR[90,1] + -17.623;
   1:  PR[91,2] = PR[90,2] + 19.393;
   1:L PR[91] R[100]mm/sec CNT100;
   1:  PR[91,1] = PR[90,1] + -20.933;
   1:  PR[91,2] = PR[90,2] + 19.218;
   1:L PR[91] R[100]mm/sec CNT100;
   1:  PR[91,1] = PR[90,1] + -24.493;
   1:  PR[91,2] = PR[90,2] + 18.487;
   1:L PR[91] R[100]mm/sec CNT100;
   1:  PR[91,1] = PR[90,1] + -27.043;
   1:  PR[91,2] = PR[90,2] + 17.561;
   1:L PR[91] R[100]mm/sec CNT100;
   1:  PR[91,1] = PR[90,1] + -28.228;
   1:  PR[91,2] = PR[90,2] + 16.962;
   1:L PR[91] R[100]mm/sec CNT100;
   1:  PR[91,1] = PR[90,1] + -30.293;
   1:  PR[91,2] = PR[90,2] + 15.817;
   1:L PR[91] R[100]mm/sec CNT100;
   1:  PR[91,1] = PR[90,1] + -31.942;
   1:  PR[91,2] = PR[90,2] + 14.426;
   1:L PR[91] R[100]mm/sec CNT100;
   1:  PR[91,1] = PR[90,1] + -33.508;
   1:  PR[91,2] = PR[90,2] + 13.187;
   1:L PR[91] R[100]mm/sec CNT100;
   1:  PR[91,1] = PR[90,1] + -34.483;
   1:  PR[91,2] = PR[90,2] + 12.138;
   1:L PR[91] R[100]mm/sec CNT100;
   1:  PR[91,1] = PR[90,1] + -36.170;
   1:  PR[91,2] = PR[90,2] + 9.783;
   1:L PR[91] R[100]mm/sec CNT100;
   1:  PR[91,1] = PR[90,1] + -36.854;
   1:  PR[91,2] = PR[90,2] + 8.743;
   1:L PR[91] R[100]mm/sec CNT100;
   1:  PR[91,1] = PR[90,1] + -37.298;
   1:  PR[91,2] = PR[90,2] + 7.745;
   1:L PR[91] R[100]mm/sec CNT100;
   1:  PR[91,1] = PR[90,1] + -38.498;
   1:  PR[91,2] = PR[90,2] + 4.758;
   1:L PR[91] R[100]mm/sec CNT100;
   1:  PR[91,1] = PR[90,1] + -38.706;
   1:  PR[91,2] = PR[90,2] + 3.951;
   1:L PR[91] R[100]mm/sec CNT100;
   1:  PR[91,1] = PR[90,1] + -39.150;
   1:  PR[91,2] = PR[90,2] + 0.453;
   1:L PR[91] R[100]mm/sec CNT100;
   1:  PR[91,1] = PR[90,1] + -39.207;
   1:  PR[91,2] = PR[90,2] + -0.277;
   1:L PR[91] R[100]mm/sec CNT100;
   1:  PR[91,1] = PR[90,1] + -38.768;
   1:  PR[91,2] = PR[90,2] + -3.707;
   1:L PR[91] R[100]mm/sec CNT100;
   1:  PR[91,1] = PR[90,1] + -38.698;
   1:  PR[91,2] = PR[90,2] + -4.608;
   1:L PR[91] R[100]mm/sec CNT100;
   1:  PR[91,1] = PR[90,1] + -38.498;
   1:  PR[91,2] = PR[90,2] + -5.382;
   1:L PR[91] R[100]mm/sec CNT100;
   1:  PR[91,1] = PR[90,1] + -37.298;
   1:  PR[91,2] = PR[90,2] + -8.369;
   1:L PR[91] R[100]mm/sec CNT100;
   1:  PR[91,1] = PR[90,1] + -36.866;
   1:  PR[91,2] = PR[90,2] + -9.338;
   1:L PR[91] R[100]mm/sec CNT100;
   1:  PR[91,1] = PR[90,1] + -35.185;
   1:  PR[91,2] = PR[90,2] + -11.672;
   1:L PR[91] R[100]mm/sec CNT100;
   1:  PR[91,1] = PR[90,1] + -34.460;
   1:  PR[91,2] = PR[90,2] + -12.786;
   1:L PR[91] R[100]mm/sec CNT100;
   1:  PR[91,1] = PR[90,1] + -33.492;
   1:  PR[91,2] = PR[90,2] + -13.829;
   1:L PR[91] R[100]mm/sec CNT100;
   1:  PR[91,1] = PR[90,1] + -31.736;
   1:  PR[91,2] = PR[90,2] + -15.318;
   1:L PR[91] R[100]mm/sec CNT100;
   1:  PR[91,1] = PR[90,1] + -30.316;
   1:  PR[91,2] = PR[90,2] + -16.428;
   1:L PR[91] R[100]mm/sec CNT100;
   1:  PR[91,1] = PR[90,1] + -28.228;
   1:  PR[91,2] = PR[90,2] + -17.586;
   1:L PR[91] R[100]mm/sec CNT100;
   1:  PR[91,1] = PR[90,1] + -27.043;
   1:  PR[91,2] = PR[90,2] + -18.185;
   1:L PR[91] R[100]mm/sec CNT100;
   1:  PR[91,1] = PR[90,1] + -24.471;
   1:  PR[91,2] = PR[90,2] + -19.119;
   1:L PR[91] R[100]mm/sec CNT100;
   1:  PR[91,1] = PR[90,1] + -24.001;
   1:  PR[91,2] = PR[90,2] + -19.232;
   1:L PR[91] R[100]mm/sec CNT100;
   1:  PR[91,1] = PR[90,1] + -21.022;
   1:  PR[91,2] = PR[90,2] + -19.832;
   1:L PR[91] R[100]mm/sec CNT100;
   1:  PR[91,1] = PR[90,1] + -17.593;
   1:  PR[91,2] = PR[90,2] + -20.018;
   1:L PR[91] R[100]mm/sec CNT100;
   1:  PR[91,1] = PR[90,1] + -14.573;
   1:  PR[91,2] = PR[90,2] + -19.714;
   1:L PR[91] R[100]mm/sec CNT100;
   1:  PR[91,1] = PR[90,1] + -13.934;
   1:  PR[91,2] = PR[90,2] + -19.625;
   1:L PR[91] R[100]mm/sec CNT100;
   1:  PR[91,1] = PR[90,1] + -11.131;
   1:  PR[91,2] = PR[90,2] + -18.900;
   1:L PR[91] R[100]mm/sec CNT100;
   1:  PR[91,1] = PR[90,1] + -7.545;
   1:  PR[91,2] = PR[90,2] + -17.342;
   1:L PR[91] R[100]mm/sec CNT100;
   1:  PR[91,1] = PR[90,1] + -5.422;
   1:  PR[91,2] = PR[90,2] + -15.984;
   1:L PR[91] R[100]mm/sec CNT100;
   1:  PR[91,1] = PR[90,1] + -5.084;
   1:  PR[91,2] = PR[90,2] + -15.740;
   1:L PR[91] R[100]mm/sec CNT100;
   1:  PR[91,1] = PR[90,1] + -3.847;
   1:  PR[91,2] = PR[90,2] + -14.658;
   1:L PR[91] R[100]mm/sec CNT100;
   1:  PR[91,1] = PR[90,1] + -2.979;
   1:  PR[91,2] = PR[90,2] + -13.875;
   1:L PR[91] R[100]mm/sec CNT100;
   1:  PR[91,1] = PR[90,1] + -2.138;
   1:  PR[91,2] = PR[90,2] + -12.889;
   1:L PR[91] R[100]mm/sec CNT100;
   1:  PR[91,1] = PR[90,1] + -1.752;
   1:  PR[91,2] = PR[90,2] + -12.580;
   1:L PR[91] R[100]mm/sec CNT100;
   1:  PR[91,1] = PR[90,1] + -0.525;
   1:  PR[91,2] = PR[90,2] + -11.712;
   1:L PR[91] R[100]mm/sec CNT100;
   1:  PR[91,1] = PR[90,1] + 0.316;
   1:  PR[91,2] = PR[90,2] + -12.011;
   1:L PR[91] R[100]mm/sec CNT100;
   1:  PR[91,1] = PR[90,1] + 1.168;
   1:L PR[91] R[100]mm/sec CNT100;
   1:  PR[91,1] = PR[90,1] + 1.737;
   1:  PR[91,2] = PR[90,2] + -12.477;
   1:L PR[91] R[100]mm/sec CNT100;
   1:  PR[91,1] = PR[90,1] + 2.275;
   1:  PR[91,2] = PR[90,2] + -12.859;
   1:L PR[91] R[100]mm/sec CNT100;
   1:  PR[91,1] = PR[90,1] + 3.148;
   1:  PR[91,2] = PR[90,2] + -13.886;
   1:L PR[91] R[100]mm/sec CNT100;
   1:  PR[91,1] = PR[90,1] + 4.015;
   1:  PR[91,2] = PR[90,2] + -14.668;
   1:L PR[91] R[100]mm/sec CNT100;
   1:  PR[91,1] = PR[90,1] + 5.225;
   1:  PR[91,2] = PR[90,2] + -15.728;
   1:L PR[91] R[100]mm/sec CNT100;
   1:  PR[91,1] = PR[90,1] + 7.196;
   1:  PR[91,2] = PR[90,2] + -16.991;
   1:L PR[91] R[100]mm/sec CNT100;
   1:  PR[91,1] = PR[90,1] + 7.721;
   1:  PR[91,2] = PR[90,2] + -17.352;
   1:L PR[91] R[100]mm/sec CNT100;
   1:  PR[91,1] = PR[90,1] + 11.280;
   1:  PR[91,2] = PR[90,2] + -18.895;
   1:L PR[91] R[100]mm/sec CNT100;
   1:  PR[91,1] = PR[90,1] + 14.063;
   1:  PR[91,2] = PR[90,2] + -19.617;
   1:L PR[91] R[100]mm/sec CNT100;
   1:  PR[91,1] = PR[90,1] + 17.421;
   1:  PR[91,2] = PR[90,2] + -19.969;
   1:L PR[91] R[100]mm/sec CNT100;
   1:  PR[91,1] = PR[90,1] + 17.768;
   1:  PR[91,2] = PR[90,2] + -20.017;
   1:L PR[91] R[100]mm/sec CNT100;
   1:  PR[91,1] = PR[90,1] + 21.063;
   1:  PR[91,2] = PR[90,2] + -19.846;
   1:L PR[91] R[100]mm/sec CNT100;
   1:  PR[91,1] = PR[90,1] + 24.625;
   1:  PR[91,2] = PR[90,2] + -19.116;
   1:L PR[91] R[100]mm/sec CNT100;
   1:  PR[91,1] = PR[90,1] + 27.186;
   1:  PR[91,2] = PR[90,2] + -18.191;
   1:L PR[91] R[100]mm/sec CNT100;
   1:  PR[91,1] = PR[90,1] + 28.369;
   1:  PR[91,2] = PR[90,2] + -17.594;
   1:L PR[91] R[100]mm/sec CNT100;
   1:  PR[91,1] = PR[90,1] + 30.431;
   1:  PR[91,2] = PR[90,2] + -16.457;
   1:L PR[91] R[100]mm/sec CNT100;
   1:  PR[91,1] = PR[90,1] + 32.078;
   1:  PR[91,2] = PR[90,2] + -15.066;
   1:L PR[91] R[100]mm/sec CNT100;
   1:  PR[91,1] = PR[90,1] + 33.640;
   1:  PR[91,2] = PR[90,2] + -13.833;
   1:L PR[91] R[100]mm/sec CNT100;
   1:  PR[91,1] = PR[90,1] + 34.622;
   1:  PR[91,2] = PR[90,2] + -12.778;
   1:L PR[91] R[100]mm/sec CNT100;
   1:  PR[91,1] = PR[90,1] + 36.310;
   1:  PR[91,2] = PR[90,2] + -10.421;
   1:L PR[91] R[100]mm/sec CNT100;
   1:  PR[91,1] = PR[90,1] + 37.008;
   1:  PR[91,2] = PR[90,2] + -9.366;
   1:L PR[91] R[100]mm/sec CNT100;
   1:  PR[91,1] = PR[90,1] + 37.451;
   1:  PR[91,2] = PR[90,2] + -8.384;
   1:L PR[91] R[100]mm/sec CNT100;
   1:  PR[91,1] = PR[90,1] + 38.650;
   1:  PR[91,2] = PR[90,2] + -5.412;
   1:L PR[91] R[100]mm/sec CNT100;
   1:  PR[91,1] = PR[90,1] + 38.859;
   1:  PR[91,2] = PR[90,2] + -4.616;
   1:L PR[91] R[100]mm/sec CNT100;
   1:  PR[91,1] = PR[90,1] + 39.303;
   1:  PR[91,2] = PR[90,2] + -1.104;
   1:L PR[91] R[100]mm/sec CNT100;
   1:  PR[91,1] = PR[90,1] + 39.364;
   1:  PR[91,2] = PR[90,2] + -0.345;
   1:L PR[91] R[100]mm/sec CNT100;
   1:  PR[91,1] = PR[90,1] + 38.925;
   1:  PR[91,2] = PR[90,2] + 3.096;
   1:L PR[91] R[100]mm/sec CNT100;
   1:  PR[91,1] = PR[90,1] + 38.850;
   1:  PR[91,2] = PR[90,2] + 4.025;
   1:L PR[91] R[100]mm/sec CNT100;
   1:  PR[91,1] = PR[90,1] + 38.650;
   1:  PR[91,2] = PR[90,2] + 4.789;
   1:L PR[91] R[100]mm/sec CNT100;
   1:  PR[91,1] = PR[90,1] + 37.450;
   1:  PR[91,2] = PR[90,2] + 7.761;
   1:L PR[91] R[100]mm/sec CNT100;
   1:  PR[91,1] = PR[90,1] + 37.019;
   1:  PR[91,2] = PR[90,2] + 8.717;
   1:L PR[91] R[100]mm/sec CNT100;
   1:  PR[91,1] = PR[90,1] + 35.335;
   1:  PR[91,2] = PR[90,2] + 11.055;
   1:L PR[91] R[100]mm/sec CNT100;
   1:  PR[91,1] = PR[90,1] + 34.600;
   1:  PR[91,2] = PR[90,2] + 12.178;
   1:L PR[91] R[100]mm/sec CNT100;
   1:  PR[91,1] = PR[90,1] + 33.621;
   1:  PR[91,2] = PR[90,2] + 13.230;
   1:L PR[91] R[100]mm/sec CNT100;
   1:  PR[91,1] = PR[90,1] + 31.866;
   1:  PR[91,2] = PR[90,2] + 14.721;
   1:L PR[91] R[100]mm/sec CNT100;
   1:  PR[91,1] = PR[90,1] + 30.454;
   1:  PR[91,2] = PR[90,2] + 15.820;
   1:L PR[91] R[100]mm/sec CNT100;
   1:  PR[91,1] = PR[90,1] + 28.367;
   1:  PR[91,2] = PR[90,2] + 16.971;
   1:L PR[91] R[100]mm/sec CNT100;
   1:  PR[91,1] = PR[90,1] + 27.184;
   1:  PR[91,2] = PR[90,2] + 17.567;
   1:L PR[91] R[100]mm/sec CNT100;
   1:  PR[91,1] = PR[90,1] + 24.601;
   1:  PR[91,2] = PR[90,2] + 18.501;
   1:L PR[91] R[100]mm/sec CNT100;
   1:  PR[91,1] = PR[90,1] + 24.135;
   1:  PR[91,2] = PR[90,2] + 18.613;
   1:L PR[91] R[100]mm/sec CNT100;
   1:  PR[91,1] = PR[90,1] + 21.156;
   1:  PR[91,2] = PR[90,2] + 19.212;
   1:L PR[91] R[100]mm/sec CNT100;
   1:  PR[91,1] = PR[90,1] + 17.743;
   1:  PR[91,2] = PR[90,2] + 19.395;
   1:L PR[91] R[100]mm/sec CNT100;
   1:  PR[91,1] = PR[90,1] + 14.732;
   1:  PR[91,2] = PR[90,2] + 19.089;
   1:L PR[91] R[100]mm/sec CNT100;
   1:  PR[91,1] = PR[90,1] + 14.093;
   1:  PR[91,2] = PR[90,2] + 19.001;
   1:L PR[91] R[100]mm/sec CNT100;
   1:  PR[91,1] = PR[90,1] + 11.291;
   1:  PR[91,2] = PR[90,2] + 18.274;
   1:L PR[91] R[100]mm/sec CNT100;
   1:  PR[91,1] = PR[90,1] + 8.834;
   1:  PR[91,2] = PR[90,2] + 17.199;
   1:L PR[91] R[100]mm/sec CNT100;
   1:  PR[91,1] = PR[90,1] + 7.725;
   1:  PR[91,2] = PR[90,2] + 16.736;
   1:L PR[91] R[100]mm/sec CNT100;
   1:  PR[91,1] = PR[90,1] + 5.607;
   1:  PR[91,2] = PR[90,2] + 15.384;
   1:L PR[91] R[100]mm/sec CNT100;
   1:  PR[91,1] = PR[90,1] + 5.391;
   1:  PR[91,2] = PR[90,2] + 15.235;
   1:L PR[91] R[100]mm/sec CNT100;
   1:  PR[91,1] = PR[90,1] + 4.980;
   1:  PR[91,2] = PR[90,2] + 14.909;
   1:L PR[91] R[100]mm/sec CNT100;
   1:  PR[91,1] = PR[90,1] + 3.232;
   1:  PR[91,2] = PR[90,2] + 13.345;
   1:L PR[91] R[100]mm/sec CNT100;
   1:  PR[91,1] = PR[90,1] + 2.501;
   1:  PR[91,2] = PR[90,2] + 12.576;
   1:L PR[91] R[100]mm/sec CNT100;
   1:  PR[91,1] = PR[90,1] + 2.136;
   1:  PR[91,2] = PR[90,2] + 12.113;
   1:L PR[91] R[100]mm/sec CNT100;
   1:  PR[91,1] = PR[90,1] + 1.418;
   1:  PR[91,2] = PR[90,2] + 11.604;
   1:L PR[91] R[100]mm/sec CNT100;
   1:  PR[91,1] = PR[90,1] + 0.780;
   1:  PR[91,2] = PR[90,2] + 11.255;
   1:L PR[91] R[100]mm/sec CNT100;
   1:  PR[91,1] = PR[90,1] + -0.611;
   1:L PR[91] R[100]mm/sec CNT100;
   1:  PR[91] = PR[90];
   1:  PR[91,1] = PR[90,1] + -1.502;
   1:  PR[91,2] = PR[90,2] + 11.977;
   1:  PR[91,3] = PR[90,3] + 27.755;
   1:L PR[91] R[100]mm/sec CNT100;
   1:  PR[91,1] = PR[90,1] + -1.800;
   1:  PR[91,2] = PR[90,2] + 12.366;
   1:L PR[91] R[100]mm/sec CNT100;
   1:  PR[91,1] = PR[90,1] + -2.127;
   1:  PR[91,2] = PR[90,2] + 12.673;
   1:L PR[91] R[100]mm/sec CNT100;
   1:  PR[91,1] = PR[90,1] + -2.870;
   1:  PR[91,2] = PR[90,2] + 13.451;
   1:L PR[91] R[100]mm/sec CNT100;
   1:  PR[91,1] = PR[90,1] + -4.523;
   1:  PR[91,2] = PR[90,2] + 14.927;
   1:L PR[91] R[100]mm/sec CNT100;
   1:  PR[91,1] = PR[90,1] + -4.983;
   1:  PR[91,2] = PR[90,2] + 15.290;
   1:L PR[91] R[100]mm/sec CNT100;
   1:  PR[91,1] = PR[90,1] + -7.298;
   1:  PR[91,2] = PR[90,2] + 16.786;
   1:L PR[91] R[100]mm/sec CNT100;
   1:  PR[91,1] = PR[90,1] + -9.793;
   1:  PR[91,2] = PR[90,2] + 17.877;
   1:L PR[91] R[100]mm/sec CNT100;
   1:  PR[91,1] = PR[90,1] + -10.935;
   1:  PR[91,2] = PR[90,2] + 18.355;
   1:L PR[91] R[100]mm/sec CNT100;
   1:  PR[91,1] = PR[90,1] + -13.591;
   1:  PR[91,2] = PR[90,2] + 19.042;
   1:L PR[91] R[100]mm/sec CNT100;
   1:  PR[91,1] = PR[90,1] + -16.804;
   1:  PR[91,2] = PR[90,2] + 19.376;
   1:L PR[91] R[100]mm/sec CNT100;
   1:  PR[91,1] = PR[90,1] + -17.398;
   1:  PR[91,2] = PR[90,2] + 19.457;
   1:L PR[91] R[100]mm/sec CNT100;
   1:  PR[91,1] = PR[90,1] + -20.627;
   1:  PR[91,2] = PR[90,2] + 19.287;
   1:L PR[91] R[100]mm/sec CNT100;
   1:  PR[91,1] = PR[90,1] + -20.849;
   1:  PR[91,2] = PR[90,2] + 19.261;
   1:L PR[91] R[100]mm/sec CNT100;
   1:  PR[91,1] = PR[90,1] + -24.103;
   1:  PR[91,2] = PR[90,2] + 18.585;
   1:L PR[91] R[100]mm/sec CNT100;
   1:  PR[91,1] = PR[90,1] + -27.017;
   1:  PR[91,2] = PR[90,2] + 17.527;
   1:L PR[91] R[100]mm/sec CNT100;
   1:  PR[91,1] = PR[90,1] + -27.677;
   1:  PR[91,2] = PR[90,2] + 17.193;
   1:L PR[91] R[100]mm/sec CNT100;
   1:  PR[91,1] = PR[90,1] + -30.109;
   1:  PR[91,2] = PR[90,2] + 15.845;
   1:L PR[91] R[100]mm/sec CNT100;
   1:  PR[91,1] = PR[90,1] + -31.292;
   1:  PR[91,2] = PR[90,2] + 14.847;
   1:L PR[91] R[100]mm/sec CNT100;
   1:  PR[91,1] = PR[90,1] + -33.200;
   1:  PR[91,2] = PR[90,2] + 13.337;
   1:L PR[91] R[100]mm/sec CNT100;
   1:  PR[91,1] = PR[90,1] + -34.407;
   1:  PR[91,2] = PR[90,2] + 12.039;
   1:L PR[91] R[100]mm/sec CNT100;
   1:  PR[91,1] = PR[90,1] + -35.794;
   1:  PR[91,2] = PR[90,2] + 10.103;
   1:L PR[91] R[100]mm/sec CNT100;
   1:  PR[91,1] = PR[90,1] + -36.677;
   1:  PR[91,2] = PR[90,2] + 8.760;
   1:L PR[91] R[100]mm/sec CNT100;
   1:  PR[91,1] = PR[90,1] + -37.252;
   1:  PR[91,2] = PR[90,2] + 7.468;
   1:L PR[91] R[100]mm/sec CNT100;
   1:  PR[91,1] = PR[90,1] + -38.280;
   1:  PR[91,2] = PR[90,2] + 4.908;
   1:L PR[91] R[100]mm/sec CNT100;
   1:  PR[91,1] = PR[90,1] + -38.567;
   1:  PR[91,2] = PR[90,2] + 3.797;
   1:L PR[91] R[100]mm/sec CNT100;
   1:  PR[91,1] = PR[90,1] + -38.950;
   1:  PR[91,2] = PR[90,2] + 0.776;
   1:L PR[91] R[100]mm/sec CNT100;
   1:  PR[91,1] = PR[90,1] + -39.033;
   1:  PR[91,2] = PR[90,2] + -0.277;
   1:L PR[91] R[100]mm/sec CNT100;
   1:  PR[91,1] = PR[90,1] + -38.653;
   1:  PR[91,2] = PR[90,2] + -3.247;
   1:L PR[91] R[100]mm/sec CNT100;
   1:  PR[91,1] = PR[90,1] + -38.559;
   1:  PR[91,2] = PR[90,2] + -4.454;
   1:L PR[91] R[100]mm/sec CNT100;
   1:  PR[91,1] = PR[90,1] + -38.280;
   1:  PR[91,2] = PR[90,2] + -5.532;
   1:L PR[91] R[100]mm/sec CNT100;
   1:  PR[91,1] = PR[90,1] + -37.252;
   1:  PR[91,2] = PR[90,2] + -8.092;
   1:L PR[91] R[100]mm/sec CNT100;
   1:  PR[91,1] = PR[90,1] + -36.689;
   1:  PR[91,2] = PR[90,2] + -9.355;
   1:L PR[91] R[100]mm/sec CNT100;
   1:  PR[91,1] = PR[90,1] + -35.270;
   1:  PR[91,2] = PR[90,2] + -11.324;
   1:L PR[91] R[100]mm/sec CNT100;
